LIN {X 0,Y 517.674,Z 1252.687,A -85,B 0,C 180,E1 12065.696,E2 12065.696} C_VEL
LIN {X 0,Y 518.294,Z 1242.725,A -85,B 0,C 180,E1 12070.089,E2 12070.089} C_VEL
LIN {X 0,Y 519.672,Z 1227.061,A -85,B 0,C 180,E1 12074.336,E2 12074.336} C_VEL
LIN {X 0,Y 522.079,Z 1206.878,A -85,B 0,C 180,E1 12078.165,E2 12078.165} C_VEL
LIN {X 0,Y 525.156,Z 1182.716,A -85,B 0,C 180,E1 12081.57,E2 12081.57} C_VEL
LIN {X 0,Y 529.072,Z 1152.709,A -85,B 0,C 180,E1 12084.747,E2 12084.747} C_VEL
LIN {X 0,Y 533.272,Z 1118.155,A -85,B 0,C 180,E1 12087.469,E2 12087.469} C_VEL
LIN {X 0,Y 537.249,Z 1080.299,A -85,B 0,C 180,E1 12089.617,E2 12089.617} C_VEL
LIN {X 0,Y 540.035,Z 1039.368,A -85,B 0,C 180,E1 12091.243,E2 12091.243} C_VEL
LIN {X 0,Y 532.268,Z 1011.624,A -85,B 0,C 180,E1 12092.744,E2 12092.744} C_VEL
LIN {X 0,Y 521.045,Z 988.142,A -85,B 0,C 180,E1 12094.497,E2 12094.497} C_VEL
LIN {X 0,Y 515.944,Z 978.381,A -85,B 0,C 180,E1 12095.418,E2 12095.418} C_VEL
LIN {X 0,Y 515.906,Z 977.53,A -85,B 0,C 180,E1 12095.954,E2 12095.954} C_VEL
LIN {X 0,Y 515.706,Z 977.53,A -85,B 0,C 180,E1 12102.493,E2 12102.493} C_VEL
LIN {X 0,Y 515.702,Z 977.53,A -85,B 0,C 180,E1 12107.495,E2 12107.495} C_VEL
LIN {X 0,Y 515.966,Z 977.849,A -85,B 0,C 180,E1 12113.885,E2 12113.885} C_VEL
LIN {X 0,Y 518.775,Z 983.54,A -85,B 0,C 180,E1 12114.433,E2 12114.433} C_VEL
LIN {X 0,Y 525.544,Z 1003.125,A -85,B 0,C 180,E1 12115.774,E2 12115.774} C_VEL
LIN {X 0,Y 540.092,Z 1052.552,A -85,B 0,C 180,E1 12118.245,E2 12118.245} C_VEL
LIN {X 0,Y 536.809,Z 1095.974,A -85,B 0,C 180,E1 12119.472,E2 12119.472} C_VEL
LIN {X 0,Y 533.589,Z 1130.82,A -85,B 0,C 180,E1 12120.973,E2 12120.973} C_VEL
LIN {X 0,Y 528.491,Z 1146.473,A -85,B 0,C 180,E1 12121.634,E2 12121.634} C_VEL
LIN {X 0,Y 523.112,Z 1161.648,A -85,B 0,C 180,E1 12122.384,E2 12122.384} C_VEL
LIN {X 0,Y 518.929,Z 1197.704,A -85,B 0,C 180,E1 12125.22,E2 12125.22} C_VEL
LIN {X 0,Y 515.24,Z 1230.103,A -85,B 0,C 180,E1 12128.666,E2 12128.666} C_VEL
LIN {X 0,Y 512.446,Z 1256.091,A -85,B 0,C 180,E1 12132.365,E2 12132.365} C_VEL
LIN {X 0,Y 510.731,Z 1276.42,A -85,B 0,C 180,E1 12136.278,E2 12136.278} C_VEL
LIN {X 0,Y 509.918,Z 1290.852,A -85,B 0,C 180,E1 12140.17,E2 12140.17} C_VEL
LIN {X 0,Y 509.696,Z 1300.49,A -85,B 0,C 180,E1 12144.192,E2 12144.192} C_VEL
LIN {X 0,Y 509.653,Z 1305.171,A -85,B 0,C 180,E1 12148.304,E2 12148.304} C_VEL
LIN {X 0,Y 509.652,Z 1305.175,A -85,B 0,C 180,E1 12151.712,E2 12151.712} C_VEL
LIN {X 0,Y 509.706,Z 1300.635,A -85,B 0,C 180,E1 12155.817,E2 12155.817} C_VEL
LIN {X 0,Y 509.891,Z 1291.146,A -85,B 0,C 180,E1 12159.847,E2 12159.847} C_VEL
LIN {X 0,Y 510.92,Z 1274.891,A -85,B 0,C 180,E1 12164.171,E2 12164.171} C_VEL
LIN {X 0,Y 512.738,Z 1253.925,A -85,B 0,C 180,E1 12168.086,E2 12168.086} C_VEL
LIN {X 0,Y 515.486,Z 1228.889,A -85,B 0,C 180,E1 12171.566,E2 12171.566} C_VEL
LIN {X 0,Y 518.975,Z 1198.242,A -85,B 0,C 180,E1 12174.779,E2 12174.779} C_VEL
LIN {X 0,Y 522.964,Z 1163.212,A -85,B 0,C 180,E1 12177.511,E2 12177.511} C_VEL
LIN {X 0,Y 526.968,Z 1123.902,A -85,B 0,C 180,E1 12179.713,E2 12179.713} C_VEL
LIN {X 0,Y 530.27,Z 1082.204,A -85,B 0,C 180,E1 12181.246,E2 12181.246} C_VEL
LIN {X 0,Y 531.189,Z 1051.195,A -85,B 0,C 180,E1 12181.983,E2 12181.983} C_VEL
LIN {X 0,Y 517.798,Z 1008.08,A -85,B 0,C 180,E1 12183.613,E2 12183.613} C_VEL
LIN {X 0,Y 514.673,Z 999.311,A -85,B 0,C 180,E1 12184.192,E2 12184.192} C_VEL
LIN {X 0,Y 508,Z 977.53,A -85,B 0,C 180,E1 12186.479,E2 12186.479} C_VEL
LIN {X 0,Y 507.893,Z 977.53,A -85,B 0,C 180,E1 12193.34,E2 12193.34} C_VEL
LIN {X 0,Y 507.84,Z 977.53,A -85,B 0,C 180,E1 12198.994,E2 12198.994} C_VEL
LIN {X 0,Y 507.949,Z 977.53,A -85,B 0,C 180,E1 12205.493,E2 12205.493} C_VEL
LIN {X 0,Y 508.183,Z 977.53,A -85,B 0,C 180,E1 12211.523,E2 12211.523} C_VEL
LIN {X 0,Y 508.423,Z 977.53,A -85,B 0,C 180,E1 12217.523,E2 12217.523} C_VEL
LIN {X 0,Y 508.509,Z 977.53,A -85,B 0,C 180,E1 12222.678,E2 12222.678} C_VEL
LIN {X 0,Y 508.671,Z 977.53,A -85,B 0,C 180,E1 12227.331,E2 12227.331} C_VEL
LIN {X 0,Y 523.418,Z 1014.68,A -85,B 0,C 180,E1 12229.87,E2 12229.87} C_VEL
LIN {X 0,Y 525.734,Z 1025.014,A -85,B 0,C 180,E1 12230.378,E2 12230.378} C_VEL
LIN {X 0,Y 522.592,Z 1078.23,A -85,B 0,C 180,E1 12231.992,E2 12231.992} C_VEL
LIN {X 0,Y 520.54,Z 1106.529,A -85,B 0,C 180,E1 12233.536,E2 12233.536} C_VEL
LIN {X 0,Y 517.847,Z 1132.303,A -85,B 0,C 180,E1 12235.712,E2 12235.712} C_VEL
LIN {X 0,Y 515.412,Z 1152.921,A -85,B 0,C 180,E1 12238.328,E2 12238.328} C_VEL
LIN {X 0,Y 513.42,Z 1168.559,A -85,B 0,C 180,E1 12241.28,E2 12241.28} C_VEL
LIN {X 0,Y 511.998,Z 1178.408,A -85,B 0,C 180,E1 12244.255,E2 12244.255} C_VEL
LIN {X 0,Y 511.229,Z 1182.945,A -85,B 0,C 180,E1 12246.82,E2 12246.82} C_VEL
LIN {X 0,Y 510.828,Z 1183.897,A -85,B 0,C 180,E1 12250.263,E2 12250.263} C_VEL
LIN {X 0,Y 511.052,Z 1178.841,A -85,B 0,C 180,E1 12253.732,E2 12253.732} C_VEL
LIN {X 0,Y 511.596,Z 1169.023,A -85,B 0,C 180,E1 12256.795,E2 12256.795} C_VEL
LIN {X 0,Y 512.738,Z 1152.99,A -85,B 0,C 180,E1 12259.878,E2 12259.878} C_VEL
LIN {X 0,Y 514.329,Z 1132.205,A -85,B 0,C 180,E1 12262.529,E2 12262.529} C_VEL
LIN {X 0,Y 515.926,Z 1107.861,A -85,B 0,C 180,E1 12264.663,E2 12264.663} C_VEL
LIN {X 0,Y 517.508,Z 1079.704,A -85,B 0,C 180,E1 12266.286,E2 12266.286} C_VEL
LIN {X 0,Y 518.405,Z 1049.368,A -85,B 0,C 180,E1 12267.293,E2 12267.293} C_VEL
LIN {X 0,Y 518.622,Z 1015.217,A -85,B 0,C 180,E1 12268.017,E2 12268.017} C_VEL
LIN {X 0,Y 508.273,Z 977.53,A -85,B 0,C 180,E1 12269.286,E2 12269.286} C_VEL
LIN {X 0,Y 507.992,Z 977.53,A -85,B 0,C 180,E1 12274.533,E2 12274.533} C_VEL
LIN {X 0,Y 507.906,Z 977.53,A -85,B 0,C 180,E1 12281.031,E2 12281.031} C_VEL
LIN {X 0,Y 507.88,Z 977.53,A -85,B 0,C 180,E1 12286.659,E2 12286.659} C_VEL
LIN {X 0,Y 507.922,Z 977.53,A -85,B 0,C 180,E1 12293.36,E2 12293.36} C_VEL
LIN {X 0,Y 508.127,Z 977.53,A -85,B 0,C 180,E1 12299.872,E2 12299.872} C_VEL
LIN {X 0,Y 508.284,Z 977.53,A -85,B 0,C 180,E1 12305.323,E2 12305.323} C_VEL
LIN {X 0,Y 508.485,Z 977.53,A -85,B 0,C 180,E1 12310.857,E2 12310.857} C_VEL
LIN {X 0,Y 508.621,Z 977.53,A -85,B 0,C 180,E1 12316.204,E2 12316.204} C_VEL
LIN {X 0,Y 508.884,Z 977.53,A -85,B 0,C 180,E1 12321.43,E2 12321.43} C_VEL
LIN {X 0,Y 509.137,Z 977.53,A -85,B 0,C 180,E1 12326.58,E2 12326.58} C_VEL
LIN {X 0,Y 509.259,Z 977.53,A -85,B 0,C 180,E1 12331.697,E2 12331.697} C_VEL
LIN {X 0,Y 508.941,Z 977.53,A -85,B 0,C 180,E1 12336.832,E2 12336.832} C_VEL
LIN {X 0,Y 508.71,Z 977.53,A -85,B 0,C 180,E1 12342.027,E2 12342.027} C_VEL
LIN {X 0,Y 508.514,Z 977.53,A -85,B 0,C 180,E1 12347.516,E2 12347.516} C_VEL
LIN {X 0,Y 508.315,Z 977.53,A -85,B 0,C 180,E1 12352.792,E2 12352.792} C_VEL
LIN {X 0,Y 508.162,Z 977.53,A -85,B 0,C 180,E1 12358.487,E2 12358.487} C_VEL
LIN {X 0,Y 508.026,Z 977.53,A -85,B 0,C 180,E1 12364.511,E2 12364.511} C_VEL
LIN {X 0,Y 507.876,Z 977.53,A -85,B 0,C 180,E1 12371.014,E2 12371.014} C_VEL
LIN {X 0,Y 507.861,Z 977.53,A -85,B 0,C 180,E1 12376.657,E2 12376.657} C_VEL
LIN {X 0,Y 507.925,Z 977.53,A -85,B 0,C 180,E1 12383.36,E2 12383.36} C_VEL
LIN {X 0,Y 508.032,Z 978.194,A -85,B 0,C 180,E1 12385.954,E2 12385.954} C_VEL
LIN {X 0,Y 527.737,Z 1030.087,A -85,B 0,C 180,E1 12388.197,E2 12388.197} C_VEL
LIN {X 0,Y 531.315,Z 1043.411,A -85,B 0,C 180,E1 12388.828,E2 12388.828} C_VEL
LIN {X 0,Y 528.029,Z 1082.986,A -85,B 0,C 180,E1 12390.438,E2 12390.438} C_VEL
LIN {X 0,Y 524.301,Z 1119.193,A -85,B 0,C 180,E1 12392.576,E2 12392.576} C_VEL
LIN {X 0,Y 520.228,Z 1153.562,A -85,B 0,C 180,E1 12395.352,E2 12395.352} C_VEL
LIN {X 0,Y 516.414,Z 1184.3,A -85,B 0,C 180,E1 12398.699,E2 12398.699} C_VEL
LIN {X 0,Y 513.431,Z 1209.4,A -85,B 0,C 180,E1 12402.381,E2 12402.381} C_VEL
LIN {X 0,Y 511.332,Z 1228.999,A -85,B 0,C 180,E1 12406.276,E2 12406.276} C_VEL
LIN {X 0,Y 510.227,Z 1242.925,A -85,B 0,C 180,E1 12410.157,E2 12410.157} C_VEL
LIN {X 0,Y 509.643,Z 1252.599,A -85,B 0,C 180,E1 12414.386,E2 12414.386} C_VEL
LIN {X 0,Y 509.472,Z 1256.861,A -85,B 0,C 180,E1 12418.284,E2 12418.284} C_VEL
LIN {X 0,Y 509.615,Z 1257.126,A -85,B 0,C 180,E1 12421.691,E2 12421.691} C_VEL
LIN {X 0,Y 509.798,Z 1253.133,A -85,B 0,C 180,E1 12425.784,E2 12425.784} C_VEL
LIN {X 0,Y 510.486,Z 1243.205,A -85,B 0,C 180,E1 12430.245,E2 12430.245} C_VEL
LIN {X 0,Y 511.978,Z 1227.568,A -85,B 0,C 180,E1 12434.556,E2 12434.556} C_VEL
LIN {X 0,Y 514.503,Z 1207.42,A -85,B 0,C 180,E1 12438.442,E2 12438.442} C_VEL
LIN {X 0,Y 517.774,Z 1183.304,A -85,B 0,C 180,E1 12441.893,E2 12441.893} C_VEL
LIN {X 0,Y 521.754,Z 1154.531,A -85,B 0,C 180,E1 12445.003,E2 12445.003} C_VEL
LIN {X 0,Y 526.022,Z 1121.129,A -85,B 0,C 180,E1 12447.716,E2 12447.716} C_VEL
LIN {X 0,Y 530.34,Z 1082.747,A -85,B 0,C 180,E1 12449.983,E2 12449.983} C_VEL
LIN {X 0,Y 533.531,Z 1041.642,A -85,B 0,C 180,E1 12451.665,E2 12451.665} C_VEL
LIN {X 0,Y 526.215,Z 1014.699,A -85,B 0,C 180,E1 12453.206,E2 12453.206} C_VEL
LIN {X 0,Y 515.247,Z 991.599,A -85,B 0,C 180,E1 12455.064,E2 12455.064} C_VEL
LIN {X 0,Y 508.007,Z 978.135,A -85,B 0,C 180,E1 12456.523,E2 12456.523} C_VEL
LIN {X 0,Y 507.751,Z 977.53,A -85,B 0,C 180,E1 12461.761,E2 12461.761} C_VEL
LIN {X 0,Y 507.746,Z 977.53,A -85,B 0,C 180,E1 12468.225,E2 12468.225} C_VEL
LIN {X 0,Y 508.045,Z 978.12,A -85,B 0,C 180,E1 12472.78,E2 12472.78} C_VEL
LIN {X 0,Y 510.907,Z 983.645,A -85,B 0,C 180,E1 12473.42,E2 12473.42} C_VEL
LIN {X 0,Y 516.711,Z 995.396,A -85,B 0,C 180,E1 12474.578,E2 12474.578} C_VEL
LIN {X 0,Y 529.642,Z 1040.211,A -85,B 0,C 180,E1 12477.114,E2 12477.114} C_VEL
LIN {X 0,Y 533.412,Z 1056.815,A -85,B 0,C 180,E1 12477.858,E2 12477.858} C_VEL
LIN {X 0,Y 529.842,Z 1098.874,A -85,B 0,C 180,E1 12479.135,E2 12479.135} C_VEL
LIN {X 0,Y 525.642,Z 1140.038,A -85,B 0,C 180,E1 12481.057,E2 12481.057} C_VEL
LIN {X 0,Y 523.112,Z 1161.648,A -85,B 0,C 180,E1 12482.384,E2 12482.384} C_VEL
LIN {X 0,Y 517.813,Z 1176.433,A -85,B 0,C 180,E1 12483.252,E2 12483.252} C_VEL
LIN {X 0,Y 512.524,Z 1190.574,A -85,B 0,C 180,E1 12484.236,E2 12484.236} C_VEL
LIN {X 0,Y 508.556,Z 1222.098,A -85,B 0,C 180,E1 12487.419,E2 12487.419} C_VEL
LIN {X 0,Y 505.44,Z 1248.801,A -85,B 0,C 180,E1 12490.981,E2 12490.981} C_VEL
LIN {X 0,Y 503.279,Z 1271.003,A -85,B 0,C 180,E1 12494.957,E2 12494.957} C_VEL
LIN {X 0,Y 502.25,Z 1287.239,A -85,B 0,C 180,E1 12498.997,E2 12498.997} C_VEL
LIN {X 0,Y 501.842,Z 1298.125,A -85,B 0,C 180,E1 12503.071,E2 12503.071} C_VEL
LIN {X 0,Y 501.743,Z 1303.439,A -85,B 0,C 180,E1 12506.545,E2 12506.545} C_VEL
LIN {X 0,Y 501.817,Z 1305.231,A -85,B 0,C 180,E1 12510.008,E2 12510.008} C_VEL
LIN {X 0,Y 501.751,Z 1303.45,A -85,B 0,C 180,E1 12513.471,E2 12513.471} C_VEL
LIN {X 0,Y 501.895,Z 1296.291,A -85,B 0,C 180,E1 12517.816,E2 12517.816} C_VEL
LIN {X 0,Y 502.37,Z 1284.818,A -85,B 0,C 180,E1 12521.752,E2 12521.752} C_VEL
LIN {X 0,Y 503.599,Z 1267.795,A -85,B 0,C 180,E1 12525.738,E2 12525.738} C_VEL
LIN {X 0,Y 505.82,Z 1245.102,A -85,B 0,C 180,E1 12529.593,E2 12529.593} C_VEL
LIN {X 0,Y 509.094,Z 1217.26,A -85,B 0,C 180,E1 12533.119,E2 12533.119} C_VEL
LIN {X 0,Y 513.025,Z 1185.22,A -85,B 0,C 180,E1 12536.165,E2 12536.165} C_VEL
LIN {X 0,Y 517.218,Z 1148.71,A -85,B 0,C 180,E1 12538.73,E2 12538.73} C_VEL
LIN {X 0,Y 521.122,Z 1108.432,A -85,B 0,C 180,E1 12540.705,E2 12540.705} C_VEL
LIN {X 0,Y 524.064,Z 1067.991,A -85,B 0,C 180,E1 12541.97,E2 12541.97} C_VEL
LIN {X 0,Y 524.17,Z 1053.575,A -85,B 0,C 180,E1 12542.301,E2 12542.301} C_VEL
LIN {X 0,Y 511.11,Z 1009.867,A -85,B 0,C 180,E1 12544.118,E2 12544.118} C_VEL
LIN {X 0,Y 506.989,Z 999.295,A -85,B 0,C 180,E1 12544.777,E2 12544.777} C_VEL
LIN {X 0,Y 499.999,Z 977.53,A -85,B 0,C 180,E1 12547.199,E2 12547.199} C_VEL
LIN {X 0,Y 499.992,Z 977.53,A -85,B 0,C 180,E1 12553.362,E2 12553.362} C_VEL
LIN {X 0,Y 499.925,Z 977.53,A -85,B 0,C 180,E1 12559.278,E2 12559.278} C_VEL
LIN {X 0,Y 499.99,Z 977.53,A -85,B 0,C 180,E1 12564.925,E2 12564.925} C_VEL
LIN {X 0,Y 500.282,Z 977.53,A -85,B 0,C 180,E1 12571.462,E2 12571.462} C_VEL
LIN {X 0,Y 500.418,Z 977.53,A -85,B 0,C 180,E1 12576.835,E2 12576.835} C_VEL
LIN {X 0,Y 500.589,Z 977.53,A -85,B 0,C 180,E1 12582.396,E2 12582.396} C_VEL
LIN {X 0,Y 500.704,Z 977.53,A -85,B 0,C 180,E1 12586.562,E2 12586.562} C_VEL
LIN {X 0,Y 515.66,Z 1013.787,A -85,B 0,C 180,E1 12589.264,E2 12589.264} C_VEL
LIN {X 0,Y 519.045,Z 1025.531,A -85,B 0,C 180,E1 12589.925,E2 12589.925} C_VEL
LIN {X 0,Y 515.519,Z 1080.567,A -85,B 0,C 180,E1 12591.668,E2 12591.668} C_VEL
LIN {X 0,Y 513.338,Z 1108.269,A -85,B 0,C 180,E1 12593.232,E2 12593.232} C_VEL
LIN {X 0,Y 510.608,Z 1132.606,A -85,B 0,C 180,E1 12595.332,E2 12595.332} C_VEL
LIN {X 0,Y 508.24,Z 1151.859,A -85,B 0,C 180,E1 12597.734,E2 12597.734} C_VEL
LIN {X 0,Y 506.21,Z 1166.874,A -85,B 0,C 180,E1 12600.441,E2 12600.441} C_VEL
LIN {X 0,Y 504.33,Z 1178.893,A -85,B 0,C 180,E1 12603.888,E2 12603.888} C_VEL
LIN {X 0,Y 503.389,Z 1184.19,A -85,B 0,C 180,E1 12606.927,E2 12606.927} C_VEL
LIN {X 0,Y 502.984,Z 1184.754,A -85,B 0,C 180,E1 12610.425,E2 12610.425} C_VEL
LIN {X 0,Y 503.256,Z 1179.276,A -85,B 0,C 180,E1 12613.949,E2 12613.949} C_VEL
LIN {X 0,Y 503.839,Z 1169.076,A -85,B 0,C 180,E1 12617.062,E2 12617.062} C_VEL
LIN {X 0,Y 504.987,Z 1152.489,A -85,B 0,C 180,E1 12620.197,E2 12620.197} C_VEL
LIN {X 0,Y 506.759,Z 1131.113,A -85,B 0,C 180,E1 12622.885,E2 12622.885} C_VEL
LIN {X 0,Y 508.43,Z 1106.223,A -85,B 0,C 180,E1 12625.023,E2 12625.023} C_VEL
LIN {X 0,Y 509.947,Z 1077.883,A -85,B 0,C 180,E1 12626.617,E2 12626.617} C_VEL
LIN {X 0,Y 510.834,Z 1047.342,A -85,B 0,C 180,E1 12627.591,E2 12627.591} C_VEL
LIN {X 0,Y 510.968,Z 1016.192,A -85,B 0,C 180,E1 12628.271,E2 12628.271} C_VEL
LIN {X 0,Y 500.334,Z 977.53,A -85,B 0,C 180,E1 12629.599,E2 12629.599} C_VEL
LIN {X 0,Y 500.034,Z 977.53,A -85,B 0,C 180,E1 12635.163,E2 12635.163} C_VEL
LIN {X 0,Y 500.026,Z 977.53,A -85,B 0,C 180,E1 12641.822,E2 12641.822} C_VEL
LIN {X 0,Y 499.982,Z 977.53,A -85,B 0,C 180,E1 12648.173,E2 12648.173} C_VEL
LIN {X 0,Y 500.008,Z 977.53,A -85,B 0,C 180,E1 12654.92,E2 12654.92} C_VEL
LIN {X 0,Y 500.265,Z 977.53,A -85,B 0,C 180,E1 12661.462,E2 12661.462} C_VEL
LIN {X 0,Y 500.393,Z 977.53,A -85,B 0,C 180,E1 12666.809,E2 12666.809} C_VEL
LIN {X 0,Y 500.609,Z 977.53,A -85,B 0,C 180,E1 12672.373,E2 12672.373} C_VEL
LIN {X 0,Y 500.777,Z 977.53,A -85,B 0,C 180,E1 12677.763,E2 12677.763} C_VEL
LIN {X 0,Y 501.074,Z 977.53,A -85,B 0,C 180,E1 12683.044,E2 12683.044} C_VEL
LIN {X 0,Y 501.241,Z 977.53,A -85,B 0,C 180,E1 12688.26,E2 12688.26} C_VEL
LIN {X 0,Y 501.19,Z 977.53,A -85,B 0,C 180,E1 12693.805,E2 12693.805} C_VEL
LIN {X 0,Y 500.897,Z 977.53,A -85,B 0,C 180,E1 12698.691,E2 12698.691} C_VEL
LIN {X 0,Y 500.67,Z 977.53,A -85,B 0,C 180,E1 12704.403,E2 12704.403} C_VEL
LIN {X 0,Y 500.51,Z 977.53,A -85,B 0,C 180,E1 12710.181,E2 12710.181} C_VEL
LIN {X 0,Y 500.295,Z 977.53,A -85,B 0,C 180,E1 12715.08,E2 12715.08} C_VEL
LIN {X 0,Y 500.138,Z 977.53,A -85,B 0,C 180,E1 12720.991,E2 12720.991} C_VEL
LIN {X 0,Y 499.975,Z 977.53,A -85,B 0,C 180,E1 12727.3,E2 12727.3} C_VEL
LIN {X 0,Y 499.98,Z 977.53,A -85,B 0,C 180,E1 12733.324,E2 12733.324} C_VEL
LIN {X 0,Y 499.918,Z 977.53,A -85,B 0,C 180,E1 12739.254,E2 12739.254} C_VEL
LIN {X 0,Y 500.1,Z 977.623,A -85,B 0,C 180,E1 12745.469,E2 12745.469} C_VEL
LIN {X 0,Y 519.896,Z 1030.125,A -85,B 0,C 180,E1 12747.782,E2 12747.782} C_VEL
LIN {X 0,Y 524.098,Z 1044.938,A -85,B 0,C 180,E1 12748.51,E2 12748.51} C_VEL
LIN {X 0,Y 520.714,Z 1083.85,A -85,B 0,C 180,E1 12750.125,E2 12750.125} C_VEL
LIN {X 0,Y 516.741,Z 1121.002,A -85,B 0,C 180,E1 12752.365,E2 12752.365} C_VEL
LIN {X 0,Y 512.524,Z 1155.393,A -85,B 0,C 180,E1 12755.215,E2 12755.215} C_VEL
LIN {X 0,Y 508.649,Z 1185.551,A -85,B 0,C 180,E1 12758.586,E2 12758.586} C_VEL
LIN {X 0,Y 505.597,Z 1210.485,A -85,B 0,C 180,E1 12762.325,E2 12762.325} C_VEL
LIN {X 0,Y 503.568,Z 1229.03,A -85,B 0,C 180,E1 12766.06,E2 12766.06} C_VEL
LIN {X 0,Y 502.397,Z 1243.094,A -85,B 0,C 180,E1 12770.002,E2 12770.002} C_VEL
LIN {X 0,Y 501.798,Z 1252.198,A -85,B 0,C 180,E1 12773.921,E2 12773.921} C_VEL
LIN {X 0,Y 501.579,Z 1257.214,A -85,B 0,C 180,E1 12778.257,E2 12778.257} C_VEL
LIN {X 0,Y 501.724,Z 1257.545,A -85,B 0,C 180,E1 12781.718,E2 12781.718} C_VEL
LIN {X 0,Y 501.932,Z 1253.311,A -85,B 0,C 180,E1 12786.052,E2 12786.052} C_VEL
LIN {X 0,Y 502.7,Z 1243.714,A -85,B 0,C 180,E1 12790.406,E2 12790.406} C_VEL
LIN {X 0,Y 504.275,Z 1228.116,A -85,B 0,C 180,E1 12794.783,E2 12794.783} C_VEL
LIN {X 0,Y 506.952,Z 1208.018,A -85,B 0,C 180,E1 12798.727,E2 12798.727} C_VEL
LIN {X 0,Y 510.417,Z 1183.973,A -85,B 0,C 180,E1 12802.225,E2 12802.225} C_VEL
LIN {X 0,Y 514.611,Z 1155.324,A -85,B 0,C 180,E1 12805.374,E2 12805.374} C_VEL
LIN {X 0,Y 519.16,Z 1121.878,A -85,B 0,C 180,E1 12808.136,E2 12808.136} C_VEL
LIN {X 0,Y 523.764,Z 1083.211,A -85,B 0,C 180,E1 12810.459,E2 12810.459} C_VEL
LIN {X 0,Y 526.921,Z 1042.452,A -85,B 0,C 180,E1 12812.187,E2 12812.187} C_VEL
LIN {X 0,Y 519.918,Z 1016.826,A -85,B 0,C 180,E1 12813.76,E2 12813.76} C_VEL
LIN {X 0,Y 509.535,Z 994.865,A -85,B 0,C 180,E1 12815.67,E2 12815.67} C_VEL
LIN {X 0,Y 502.475,Z 983.287,A -85,B 0,C 180,E1 12817.181,E2 12817.181} C_VEL
LIN {X 0,Y 499.956,Z 977.901,A -85,B 0,C 180,E1 12817.878,E2 12817.878} C_VEL
LIN {X 0,Y 499.824,Z 977.53,A -85,B 0,C 180,E1 12824.184,E2 12824.184} C_VEL
LIN {X 0,Y 499.892,Z 977.53,A -85,B 0,C 180,E1 12830.476,E2 12830.476} C_VEL
LIN {X 0,Y 500.005,Z 978.235,A -85,B 0,C 180,E1 12831.423,E2 12831.423} C_VEL
LIN {X 0,Y 503.017,Z 983.675,A -85,B 0,C 180,E1 12832.221,E2 12832.221} C_VEL
LIN {X 0,Y 511.284,Z 998.417,A -85,B 0,C 180,E1 12834.011,E2 12834.011} C_VEL
LIN {X 0,Y 523.258,Z 1041.663,A -85,B 0,C 180,E1 12836.591,E2 12836.591} C_VEL
LIN {X 0,Y 526.926,Z 1058.458,A -85,B 0,C 180,E1 12837.394,E2 12837.394} C_VEL
LIN {X 0,Y 523.013,Z 1100.851,A -85,B 0,C 180,E1 12838.742,E2 12838.742} C_VEL
LIN {X 0,Y 518.535,Z 1141.968,A -85,B 0,C 180,E1 12840.738,E2 12840.738} C_VEL
LIN {X 0,Y 513.979,Z 1179.263,A -85,B 0,C 180,E1 12843.292,E2 12843.292} C_VEL
LIN {X 0,Y 512.524,Z 1190.574,A -85,B 0,C 180,E1 12844.236,E2 12844.236} C_VEL
LIN {X 0,Y 507.109,Z 1204.205,A -85,B 0,C 180,E1 12845.327,E2 12845.327} C_VEL
LIN {X 0,Y 501.705,Z 1217.109,A -85,B 0,C 180,E1 12846.516,E2 12846.516} C_VEL
LIN {X 0,Y 498.124,Z 1245.562,A -85,B 0,C 180,E1 12850.228,E2 12850.228} C_VEL
LIN {X 0,Y 495.72,Z 1268.581,A -85,B 0,C 180,E1 12854.282,E2 12854.282} C_VEL
LIN {X 0,Y 494.413,Z 1286.258,A -85,B 0,C 180,E1 12858.635,E2 12858.635} C_VEL
LIN {X 0,Y 493.946,Z 1297.763,A -85,B 0,C 180,E1 12862.96,E2 12862.96} C_VEL
LIN {X 0,Y 493.856,Z 1303.072,A -85,B 0,C 180,E1 12866.49,E2 12866.49} C_VEL
LIN {X 0,Y 493.926,Z 1304.832,A -85,B 0,C 180,E1 12870.008,E2 12870.008} C_VEL
LIN {X 0,Y 493.829,Z 1302.415,A -85,B 0,C 180,E1 12874.129,E2 12874.129} C_VEL
LIN {X 0,Y 494.036,Z 1294.768,A -85,B 0,C 180,E1 12878.385,E2 12878.385} C_VEL
LIN {X 0,Y 494.733,Z 1280.939,A -85,B 0,C 180,E1 12882.838,E2 12882.838} C_VEL
LIN {X 0,Y 496.297,Z 1261.254,A -85,B 0,C 180,E1 12887.098,E2 12887.098} C_VEL
LIN {X 0,Y 498.997,Z 1237.037,A -85,B 0,C 180,E1 12890.913,E2 12890.913} C_VEL
LIN {X 0,Y 502.693,Z 1207.602,A -85,B 0,C 180,E1 12894.376,E2 12894.376} C_VEL
LIN {X 0,Y 506.726,Z 1174.921,A -85,B 0,C 180,E1 12897.26,E2 12897.26} C_VEL
LIN {X 0,Y 511.062,Z 1137.787,A -85,B 0,C 180,E1 12899.664,E2 12899.664} C_VEL
LIN {X 0,Y 514.859,Z 1096.916,A -85,B 0,C 180,E1 12901.489,E2 12901.489} C_VEL
LIN {X 0,Y 517.047,Z 1055.645,A -85,B 0,C 180,E1 12902.635,E2 12902.635} C_VEL
LIN {X 0,Y 504.776,Z 1012.446,A -85,B 0,C 180,E1 12904.605,E2 12904.605} C_VEL
LIN {X 0,Y 498.679,Z 997.453,A -85,B 0,C 180,E1 12905.61,E2 12905.61} C_VEL
LIN {X 0,Y 492.063,Z 977.53,A -85,B 0,C 180,E1 12908.026,E2 12908.026} C_VEL
LIN {X 0,Y 492.063,Z 977.53,A -85,B 0,C 180,E1 12912.657,E2 12912.657} C_VEL
LIN {X 0,Y 492.054,Z 977.53,A -85,B 0,C 180,E1 12917.665,E2 12917.665} C_VEL
LIN {X 0,Y 491.991,Z 977.53,A -85,B 0,C 180,E1 12924.205,E2 12924.205} C_VEL
LIN {X 0,Y 492.248,Z 977.53,A -85,B 0,C 180,E1 12930.512,E2 12930.512} C_VEL
LIN {X 0,Y 492.49,Z 977.53,A -85,B 0,C 180,E1 12936.44,E2 12936.44} C_VEL
LIN {X 0,Y 492.712,Z 977.53,A -85,B 0,C 180,E1 12942.459,E2 12942.459} C_VEL
LIN {X 0,Y 492.761,Z 977.613,A -85,B 0,C 180,E1 12945.725,E2 12945.725} C_VEL
LIN {X 0,Y 507.368,Z 1011.543,A -85,B 0,C 180,E1 12948.507,E2 12948.507} C_VEL
LIN {X 0,Y 512.187,Z 1028.95,A -85,B 0,C 180,E1 12949.542,E2 12949.542} C_VEL
LIN {X 0,Y 508.538,Z 1081.909,A -85,B 0,C 180,E1 12951.284,E2 12951.284} C_VEL
LIN {X 0,Y 506.127,Z 1110.036,A -85,B 0,C 180,E1 12952.919,E2 12952.919} C_VEL
LIN {X 0,Y 503.271,Z 1134.096,A -85,B 0,C 180,E1 12955.047,E2 12955.047} C_VEL
LIN {X 0,Y 500.495,Z 1154.757,A -85,B 0,C 180,E1 12957.743,E2 12957.743} C_VEL
LIN {X 0,Y 498.149,Z 1170.811,A -85,B 0,C 180,E1 12960.884,E2 12960.884} C_VEL
LIN {X 0,Y 496.368,Z 1181.461,A -85,B 0,C 180,E1 12964.389,E2 12964.389} C_VEL
LIN {X 0,Y 495.539,Z 1185.436,A -85,B 0,C 180,E1 12967.037,E2 12967.037} C_VEL
LIN {X 0,Y 495.154,Z 1185.542,A -85,B 0,C 180,E1 12970.592,E2 12970.592} C_VEL
LIN {X 0,Y 495.422,Z 1179.69,A -85,B 0,C 180,E1 12974.174,E2 12974.174} C_VEL
LIN {X 0,Y 496.17,Z 1168.057,A -85,B 0,C 180,E1 12977.563,E2 12977.563} C_VEL
LIN {X 0,Y 497.313,Z 1151.94,A -85,B 0,C 180,E1 12980.522,E2 12980.522} C_VEL
LIN {X 0,Y 499.209,Z 1129.928,A -85,B 0,C 180,E1 12983.251,E2 12983.251} C_VEL
LIN {X 0,Y 500.959,Z 1104.075,A -85,B 0,C 180,E1 12985.423,E2 12985.423} C_VEL
LIN {X 0,Y 502.468,Z 1075.953,A -85,B 0,C 180,E1 12986.958,E2 12986.958} C_VEL
LIN {X 0,Y 503.409,Z 1043.176,A -85,B 0,C 180,E1 12987.941,E2 12987.941} C_VEL
LIN {X 0,Y 503.447,Z 1017.654,A -85,B 0,C 180,E1 12988.515,E2 12988.515} C_VEL
LIN {X 0,Y 492.401,Z 977.53,A -85,B 0,C 180,E1 12989.936,E2 12989.936} C_VEL
LIN {X 0,Y 492.057,Z 977.53,A -85,B 0,C 180,E1 12996.794,E2 12996.794} C_VEL
LIN {X 0,Y 492.086,Z 977.53,A -85,B 0,C 180,E1 13002.655,E2 13002.655} C_VEL
LIN {X 0,Y 492.043,Z 977.53,A -85,B 0,C 180,E1 13007.665,E2 13007.665} C_VEL
LIN {X 0,Y 492.001,Z 977.53,A -85,B 0,C 180,E1 13014.176,E2 13014.176} C_VEL
LIN {X 0,Y 492.236,Z 977.53,A -85,B 0,C 180,E1 13020.484,E2 13020.484} C_VEL
LIN {X 0,Y 492.474,Z 977.53,A -85,B 0,C 180,E1 13026.414,E2 13026.414} C_VEL
LIN {X 0,Y 492.708,Z 977.53,A -85,B 0,C 180,E1 13032.454,E2 13032.454} C_VEL
LIN {X 0,Y 492.843,Z 977.53,A -85,B 0,C 180,E1 13037.563,E2 13037.563} C_VEL
LIN {X 0,Y 493.152,Z 977.53,A -85,B 0,C 180,E1 13042.932,E2 13042.932} C_VEL
LIN {X 0,Y 493.355,Z 977.53,A -85,B 0,C 180,E1 13048.232,E2 13048.232} C_VEL
LIN {X 0,Y 493.341,Z 977.53,A -85,B 0,C 180,E1 13053.514,E2 13053.514} C_VEL
LIN {X 0,Y 492.978,Z 977.53,A -85,B 0,C 180,E1 13058.832,E2 13058.832} C_VEL
LIN {X 0,Y 492.778,Z 977.53,A -85,B 0,C 180,E1 13064.232,E2 13064.232} C_VEL
LIN {X 0,Y 492.616,Z 977.53,A -85,B 0,C 180,E1 13069.768,E2 13069.768} C_VEL
LIN {X 0,Y 492.331,Z 977.53,A -85,B 0,C 180,E1 13075.514,E2 13075.514} C_VEL
LIN {X 0,Y 492.196,Z 977.53,A -85,B 0,C 180,E1 13081.548,E2 13081.548} C_VEL
LIN {X 0,Y 492.072,Z 977.53,A -85,B 0,C 180,E1 13088.005,E2 13088.005} C_VEL
LIN {X 0,Y 492.072,Z 977.53,A -85,B 0,C 180,E1 13092.634,E2 13092.634} C_VEL
LIN {X 0,Y 492.03,Z 977.53,A -85,B 0,C 180,E1 13097.643,E2 13097.643} C_VEL
LIN {X 0,Y 492.022,Z 977.53,A -85,B 0,C 180,E1 13104.177,E2 13104.177} C_VEL
LIN {X 0,Y 492.139,Z 977.53,A -85,B 0,C 180,E1 13104.989,E2 13104.989} C_VEL
LIN {X 0,Y 512.159,Z 1030.55,A -85,B 0,C 180,E1 13107.375,E2 13107.375} C_VEL
LIN {X 0,Y 516.773,Z 1047.714,A -85,B 0,C 180,E1 13108.232,E2 13108.232} C_VEL
LIN {X 0,Y 513.204,Z 1086.842,A -85,B 0,C 180,E1 13109.922,E2 13109.922} C_VEL
LIN {X 0,Y 509.048,Z 1124.404,A -85,B 0,C 180,E1 13112.273,E2 13112.273} C_VEL
LIN {X 0,Y 504.615,Z 1158.836,A -85,B 0,C 180,E1 13115.249,E2 13115.249} C_VEL
LIN {X 0,Y 500.682,Z 1188.432,A -85,B 0,C 180,E1 13118.694,E2 13118.694} C_VEL
LIN {X 0,Y 497.637,Z 1212.776,A -85,B 0,C 180,E1 13122.49,E2 13122.49} C_VEL
LIN {X 0,Y 495.437,Z 1232.615,A -85,B 0,C 180,E1 13126.728,E2 13126.728} C_VEL
LIN {X 0,Y 494.318,Z 1246.817,A -85,B 0,C 180,E1 13131.172,E2 13131.172} C_VEL
LIN {X 0,Y 493.791,Z 1255.09,A -85,B 0,C 180,E1 13135.537,E2 13135.537} C_VEL
LIN {X 0,Y 493.769,Z 1258.191,A -85,B 0,C 180,E1 13139.987,E2 13139.987} C_VEL
LIN {X 0,Y 493.858,Z 1256.883,A -85,B 0,C 180,E1 13143.505,E2 13143.505} C_VEL
LIN {X 0,Y 494.307,Z 1250.605,A -85,B 0,C 180,E1 13147.915,E2 13147.915} C_VEL
LIN {X 0,Y 495.488,Z 1238.763,A -85,B 0,C 180,E1 13152.347,E2 13152.347} C_VEL
LIN {X 0,Y 497.652,Z 1221.505,A -85,B 0,C 180,E1 13156.602,E2 13156.602} C_VEL
LIN {X 0,Y 500.774,Z 1199.915,A -85,B 0,C 180,E1 13160.433,E2 13160.433} C_VEL
LIN {X 0,Y 504.968,Z 1172.558,A -85,B 0,C 180,E1 13164.043,E2 13164.043} C_VEL
LIN {X 0,Y 509.998,Z 1139.291,A -85,B 0,C 180,E1 13167.292,E2 13167.292} C_VEL
LIN {X 0,Y 514.926,Z 1102.902,A -85,B 0,C 180,E1 13169.887,E2 13169.887} C_VEL
LIN {X 0,Y 519.41,Z 1064.543,A -85,B 0,C 180,E1 13171.839,E2 13171.839} C_VEL
LIN {X 0,Y 520.561,Z 1044.416,A -85,B 0,C 180,E1 13172.677,E2 13172.677} C_VEL
LIN {X 0,Y 513.932,Z 1019.448,A -85,B 0,C 180,E1 13174.306,E2 13174.306} C_VEL
LIN {X 0,Y 504.129,Z 998.823,A -85,B 0,C 180,E1 13176.273,E2 13176.273} C_VEL
LIN {X 0,Y 497.569,Z 988.1,A -85,B 0,C 180,E1 13177.813,E2 13177.813} C_VEL
LIN {X 0,Y 494.951,Z 983.678,A -85,B 0,C 180,E1 13178.57,E2 13178.57} C_VEL
LIN {X 0,Y 492.029,Z 978.397,A -85,B 0,C 180,E1 13179.589,E2 13179.589} C_VEL
LIN {X 0,Y 491.97,Z 977.53,A -85,B 0,C 180,E1 13180.278,E2 13180.278} C_VEL
LIN {X 0,Y 491.896,Z 977.53,A -85,B 0,C 180,E1 13185.089,E2 13185.089} C_VEL
LIN {X 0,Y 491.979,Z 978.308,A -85,B 0,C 180,E1 13189.643,E2 13189.643} C_VEL
LIN {X 0,Y 495.15,Z 983.796,A -85,B 0,C 180,E1 13190.748,E2 13190.748} C_VEL
LIN {X 0,Y 503.507,Z 997.303,A -85,B 0,C 180,E1 13192.889,E2 13192.889} C_VEL
LIN {X 0,Y 507.189,Z 1005.771,A -85,B 0,C 180,E1 13193.739,E2 13193.739} C_VEL
LIN {X 0,Y 518.647,Z 1050.506,A -85,B 0,C 180,E1 13196.419,E2 13196.419} C_VEL
LIN {X 0,Y 520.422,Z 1061.325,A -85,B 0,C 180,E1 13196.934,E2 13196.934} C_VEL
LIN {X 0,Y 516.021,Z 1105.004,A -85,B 0,C 180,E1 13198.417,E2 13198.417} C_VEL
LIN {X 0,Y 511.03,Z 1146.344,A -85,B 0,C 180,E1 13200.557,E2 13200.557} C_VEL
LIN {X 0,Y 506.23,Z 1183.12,A -85,B 0,C 180,E1 13203.21,E2 13203.21} C_VEL
LIN {X 0,Y 501.824,Z 1216.297,A -85,B 0,C 180,E1 13206.425,E2 13206.425} C_VEL
LIN {X 0,Y 501.705,Z 1217.109,A -85,B 0,C 180,E1 13206.516,E2 13206.516} C_VEL
LIN {X 0,Y 496.255,Z 1229.344,A -85,B 0,C 180,E1 13207.825,E2 13207.825} C_VEL
LIN {X 0,Y 491.029,Z 1240.799,A -85,B 0,C 180,E1 13209.242,E2 13209.242} C_VEL
LIN {X 0,Y 488.186,Z 1264.851,A -85,B 0,C 180,E1 13213.324,E2 13213.324} C_VEL
LIN {X 0,Y 486.712,Z 1282.415,A -85,B 0,C 180,E1 13217.421,E2 13217.421} C_VEL
LIN {X 0,Y 486.153,Z 1295.547,A -85,B 0,C 180,E1 13221.946,E2 13221.946} C_VEL
LIN {X 0,Y 485.955,Z 1302.713,A -85,B 0,C 180,E1 13226.433,E2 13226.433} C_VEL
LIN {X 0,Y 486.036,Z 1304.431,A -85,B 0,C 180,E1 13230.008,E2 13230.008} C_VEL
LIN {X 0,Y 485.942,Z 1302.104,A -85,B 0,C 180,E1 13234.067,E2 13234.067} C_VEL
LIN {X 0,Y 486.143,Z 1294.235,A -85,B 0,C 180,E1 13238.522,E2 13238.522} C_VEL
LIN {X 0,Y 486.889,Z 1280.259,A -85,B 0,C 180,E1 13243.048,E2 13243.048} C_VEL
LIN {X 0,Y 488.578,Z 1260.371,A -85,B 0,C 180,E1 13247.377,E2 13247.377} C_VEL
LIN {X 0,Y 491.41,Z 1235.909,A -85,B 0,C 180,E1 13251.251,E2 13251.251} C_VEL
LIN {X 0,Y 495.106,Z 1207.281,A -85,B 0,C 180,E1 13254.654,E2 13254.654} C_VEL
LIN {X 0,Y 499.385,Z 1173.578,A -85,B 0,C 180,E1 13257.658,E2 13257.658} C_VEL
LIN {X 0,Y 503.955,Z 1135.486,A -85,B 0,C 180,E1 13260.125,E2 13260.125} C_VEL
LIN {X 0,Y 507.823,Z 1094.549,A -85,B 0,C 180,E1 13261.93,E2 13261.93} C_VEL
LIN {X 0,Y 509.919,Z 1057.283,A -85,B 0,C 180,E1 13263.026,E2 13263.026} C_VEL
LIN {X 0,Y 499.263,Z 1016.91,A -85,B 0,C 180,E1 13265.002,E2 13265.002} C_VEL
LIN {X 0,Y 490.224,Z 995.351,A -85,B 0,C 180,E1 13266.55,E2 13266.55} C_VEL
LIN {X 0,Y 484.116,Z 977.53,A -85,B 0,C 180,E1 13268.867,E2 13268.867} C_VEL
LIN {X 0,Y 484.059,Z 977.53,A -85,B 0,C 180,E1 13273.973,E2 13273.973} C_VEL
LIN {X 0,Y 484.053,Z 977.53,A -85,B 0,C 180,E1 13278.923,E2 13278.923} C_VEL
LIN {X 0,Y 484.065,Z 977.53,A -85,B 0,C 180,E1 13284.491,E2 13284.491} C_VEL
LIN {X 0,Y 484.307,Z 977.53,A -85,B 0,C 180,E1 13289.979,E2 13289.979} C_VEL
LIN {X 0,Y 484.517,Z 977.53,A -85,B 0,C 180,E1 13296.028,E2 13296.028} C_VEL
LIN {X 0,Y 484.716,Z 977.53,A -85,B 0,C 180,E1 13301.799,E2 13301.799} C_VEL
LIN {X 0,Y 484.817,Z 977.829,A -85,B 0,C 180,E1 13304.817,E2 13304.817} C_VEL
LIN {X 0,Y 499.507,Z 1010.674,A -85,B 0,C 180,E1 13307.782,E2 13307.782} C_VEL
LIN {X 0,Y 505.541,Z 1030.595,A -85,B 0,C 180,E1 13309.082,E2 13309.082} C_VEL
LIN {X 0,Y 501.595,Z 1083.395,A -85,B 0,C 180,E1 13310.888,E2 13310.888} C_VEL
LIN {X 0,Y 499.147,Z 1110.474,A -85,B 0,C 180,E1 13312.491,E2 13312.491} C_VEL
LIN {X 0,Y 495.967,Z 1135.592,A -85,B 0,C 180,E1 13314.754,E2 13314.754} C_VEL
LIN {X 0,Y 493.108,Z 1155.623,A -85,B 0,C 180,E1 13317.417,E2 13317.417} C_VEL
LIN {X 0,Y 490.674,Z 1171.045,A -85,B 0,C 180,E1 13320.455,E2 13320.455} C_VEL
LIN {X 0,Y 488.943,Z 1181.047,A -85,B 0,C 180,E1 13323.566,E2 13323.566} C_VEL
LIN {X 0,Y 487.696,Z 1186.626,A -85,B 0,C 180,E1 13327.151,E2 13327.151} C_VEL
LIN {X 0,Y 487.318,Z 1186.329,A -85,B 0,C 180,E1 13330.764,E2 13330.764} C_VEL
LIN {X 0,Y 487.629,Z 1180.049,A -85,B 0,C 180,E1 13334.406,E2 13334.406} C_VEL
LIN {X 0,Y 488.433,Z 1167.95,A -85,B 0,C 180,E1 13337.851,E2 13337.851} C_VEL
LIN {X 0,Y 489.684,Z 1151.339,A -85,B 0,C 180,E1 13340.857,E2 13340.857} C_VEL
LIN {X 0,Y 491.52,Z 1129.603,A -85,B 0,C 180,E1 13343.524,E2 13343.524} C_VEL
LIN {X 0,Y 493.407,Z 1103.421,A -85,B 0,C 180,E1 13345.718,E2 13345.718} C_VEL
LIN {X 0,Y 494.937,Z 1074.285,A -85,B 0,C 180,E1 13347.283,E2 13347.283} C_VEL
LIN {X 0,Y 495.986,Z 1039.705,A -85,B 0,C 180,E1 13348.285,E2 13348.285} C_VEL
LIN {X 0,Y 496.041,Z 1019.546,A -85,B 0,C 180,E1 13348.753,E2 13348.753} C_VEL
LIN {X 0,Y 484.436,Z 977.53,A -85,B 0,C 180,E1 13350.283,E2 13350.283} C_VEL
LIN {X 0,Y 484.141,Z 977.53,A -85,B 0,C 180,E1 13356.499,E2 13356.499} C_VEL
LIN {X 0,Y 484.107,Z 977.53,A -85,B 0,C 180,E1 13361.293,E2 13361.293} C_VEL
LIN {X 0,Y 484.055,Z 977.53,A -85,B 0,C 180,E1 13366.463,E2 13366.463} C_VEL
LIN {X 0,Y 484.115,Z 977.53,A -85,B 0,C 180,E1 13371.501,E2 13371.501} C_VEL
LIN {X 0,Y 484.184,Z 977.53,A -85,B 0,C 180,E1 13377.848,E2 13377.848} C_VEL
LIN {X 0,Y 484.426,Z 977.53,A -85,B 0,C 180,E1 13384.02,E2 13384.02} C_VEL
LIN {X 0,Y 484.661,Z 977.53,A -85,B 0,C 180,E1 13389.876,E2 13389.876} C_VEL
LIN {X 0,Y 484.864,Z 977.53,A -85,B 0,C 180,E1 13395.673,E2 13395.673} C_VEL
LIN {X 0,Y 485.12,Z 977.53,A -85,B 0,C 180,E1 13401.007,E2 13401.007} C_VEL
LIN {X 0,Y 485.449,Z 977.53,A -85,B 0,C 180,E1 13406.413,E2 13406.413} C_VEL
LIN {X 0,Y 485.553,Z 977.53,A -85,B 0,C 180,E1 13411.78,E2 13411.78} C_VEL
LIN {X 0,Y 485.187,Z 977.53,A -85,B 0,C 180,E1 13417.168,E2 13417.168} C_VEL
LIN {X 0,Y 484.911,Z 977.53,A -85,B 0,C 180,E1 13422.626,E2 13422.626} C_VEL
LIN {X 0,Y 484.731,Z 977.53,A -85,B 0,C 180,E1 13428.207,E2 13428.207} C_VEL
LIN {X 0,Y 484.463,Z 977.53,A -85,B 0,C 180,E1 13433.982,E2 13433.982} C_VEL
LIN {X 0,Y 484.313,Z 977.53,A -85,B 0,C 180,E1 13440.029,E2 13440.029} C_VEL
LIN {X 0,Y 484.132,Z 977.53,A -85,B 0,C 180,E1 13446.479,E2 13446.479} C_VEL
LIN {X 0,Y 484.087,Z 977.53,A -85,B 0,C 180,E1 13451.291,E2 13451.291} C_VEL
LIN {X 0,Y 484.043,Z 977.53,A -85,B 0,C 180,E1 13456.462,E2 13456.462} C_VEL
LIN {X 0,Y 484.088,Z 977.53,A -85,B 0,C 180,E1 13463.496,E2 13463.496} C_VEL
LIN {X 0,Y 484.19,Z 977.825,A -85,B 0,C 180,E1 13464.505,E2 13464.505} C_VEL
LIN {X 0,Y 504.454,Z 1031.081,A -85,B 0,C 180,E1 13466.968,E2 13466.968} C_VEL
LIN {X 0,Y 509.521,Z 1049.091,A -85,B 0,C 180,E1 13467.899,E2 13467.899} C_VEL
LIN {X 0,Y 505.799,Z 1089.073,A -85,B 0,C 180,E1 13469.676,E2 13469.676} C_VEL
LIN {X 0,Y 501.294,Z 1127.569,A -85,B 0,C 180,E1 13472.174,E2 13472.174} C_VEL
LIN {X 0,Y 496.782,Z 1161.298,A -85,B 0,C 180,E1 13475.193,E2 13475.193} C_VEL
LIN {X 0,Y 492.914,Z 1189.612,A -85,B 0,C 180,E1 13478.579,E2 13478.579} C_VEL
LIN {X 0,Y 489.825,Z 1213.804,A -85,B 0,C 180,E1 13482.434,E2 13482.434} C_VEL
LIN {X 0,Y 487.659,Z 1232.608,A -85,B 0,C 180,E1 13486.512,E2 13486.512} C_VEL
LIN {X 0,Y 486.452,Z 1246.974,A -85,B 0,C 180,E1 13491.028,E2 13491.028} C_VEL
LIN {X 0,Y 485.899,Z 1255.574,A -85,B 0,C 180,E1 13495.606,E2 13495.606} C_VEL
LIN {X 0,Y 485.878,Z 1258.572,A -85,B 0,C 180,E1 13499.987,E2 13499.987} C_VEL
LIN {X 0,Y 485.976,Z 1256.974,A -85,B 0,C 180,E1 13503.964,E2 13503.964} C_VEL
LIN {X 0,Y 486.484,Z 1251.128,A -85,B 0,C 180,E1 13508.043,E2 13508.043} C_VEL
LIN {X 0,Y 487.732,Z 1239.349,A -85,B 0,C 180,E1 13512.546,E2 13512.546} C_VEL
LIN {X 0,Y 490.045,Z 1222.073,A -85,B 0,C 180,E1 13516.888,E2 13516.888} C_VEL
LIN {X 0,Y 493.433,Z 1200.309,A -85,B 0,C 180,E1 13520.81,E2 13520.81} C_VEL
LIN {X 0,Y 497.746,Z 1173.596,A -85,B 0,C 180,E1 13524.398,E2 13524.398} C_VEL
LIN {X 0,Y 502.988,Z 1141.099,A -85,B 0,C 180,E1 13527.65,E2 13527.65} C_VEL
LIN {X 0,Y 508.293,Z 1104.221,A -85,B 0,C 180,E1 13530.344,E2 13530.344} C_VEL
LIN {X 0,Y 513.155,Z 1065.355,A -85,B 0,C 180,E1 13532.366,E2 13532.366} C_VEL
LIN {X 0,Y 514.264,Z 1046.17,A -85,B 0,C 180,E1 13533.206,E2 13533.206} C_VEL
LIN {X 0,Y 508.138,Z 1022.333,A -85,B 0,C 180,E1 13534.87,E2 13534.87} C_VEL
LIN {X 0,Y 498.591,Z 1001.77,A -85,B 0,C 180,E1 13537.001,E2 13537.001} C_VEL
LIN {X 0,Y 491.402,Z 990.204,A -85,B 0,C 180,E1 13538.969,E2 13538.969} C_VEL
LIN {X 0,Y 487.815,Z 984.239,A -85,B 0,C 180,E1 13540.344,E2 13540.344} C_VEL
LIN {X 0,Y 484.109,Z 978.638,A -85,B 0,C 180,E1 13542.58,E2 13542.58} C_VEL
LIN {X 0,Y 483.926,Z 977.53,A -85,B 0,C 180,E1 13543.516,E2 13543.516} C_VEL
LIN {X 0,Y 483.977,Z 978.261,A -85,B 0,C 180,E1 13546.477,E2 13546.477} C_VEL
LIN {X 0,Y 487.927,Z 984.313,A -85,B 0,C 180,E1 13548.939,E2 13548.939} C_VEL
LIN {X 0,Y 493.762,Z 993.833,A -85,B 0,C 180,E1 13551.025,E2 13551.025} C_VEL
LIN {X 0,Y 501.573,Z 1007.116,A -85,B 0,C 180,E1 13552.999,E2 13552.999} C_VEL
LIN {X 0,Y 512.009,Z 1050.026,A -85,B 0,C 180,E1 13555.757,E2 13555.757} C_VEL
LIN {X 0,Y 514.217,Z 1062.345,A -85,B 0,C 180,E1 13556.405,E2 13556.405} C_VEL
LIN {X 0,Y 509.376,Z 1106.176,A -85,B 0,C 180,E1 13557.957,E2 13557.957} C_VEL
LIN {X 0,Y 504.068,Z 1147.297,A -85,B 0,C 180,E1 13560.15,E2 13560.15} C_VEL
LIN {X 0,Y 498.912,Z 1184.444,A -85,B 0,C 180,E1 13562.908,E2 13562.908} C_VEL
LIN {X 0,Y 494.14,Z 1218.096,A -85,B 0,C 180,E1 13566.281,E2 13566.281} C_VEL
LIN {X 0,Y 491.029,Z 1240.799,A -85,B 0,C 180,E1 13569.242,E2 13569.242} C_VEL
LIN {X 0,Y 485.994,Z 1251.489,A -85,B 0,C 180,E1 13570.764,E2 13570.764} C_VEL
LIN {X 0,Y 480.901,Z 1261.225,A -85,B 0,C 180,E1 13572.392,E2 13572.392} C_VEL
LIN {X 0,Y 479.028,Z 1280.419,A -85,B 0,C 180,E1 13576.751,E2 13576.751} C_VEL
LIN {X 0,Y 478.275,Z 1293.073,A -85,B 0,C 180,E1 13580.894,E2 13580.894} C_VEL
LIN {X 0,Y 478.121,Z 1300.151,A -85,B 0,C 180,E1 13584.553,E2 13584.553} C_VEL
LIN {X 0,Y 478.08,Z 1303.665,A -85,B 0,C 180,E1 13588.192,E2 13588.192} C_VEL
LIN {X 0,Y 478.108,Z 1303.51,A -85,B 0,C 180,E1 13591.825,E2 13591.825} C_VEL
LIN {X 0,Y 478.176,Z 1298.364,A -85,B 0,C 180,E1 13596.376,E2 13596.376} C_VEL
LIN {X 0,Y 478.454,Z 1288.769,A -85,B 0,C 180,E1 13600.501,E2 13600.501} C_VEL
LIN {X 0,Y 479.621,Z 1272.638,A -85,B 0,C 180,E1 13604.947,E2 13604.947} C_VEL
LIN {X 0,Y 481.686,Z 1252.265,A -85,B 0,C 180,E1 13608.937,E2 13608.937} C_VEL
LIN {X 0,Y 485.083,Z 1225.504,A -85,B 0,C 180,E1 13612.812,E2 13612.812} C_VEL
LIN {X 0,Y 489.142,Z 1194.524,A -85,B 0,C 180,E1 13616.167,E2 13616.167} C_VEL
LIN {X 0,Y 493.743,Z 1158.719,A -85,B 0,C 180,E1 13619.041,E2 13619.041} C_VEL
LIN {X 0,Y 498.206,Z 1119.762,A -85,B 0,C 180,E1 13621.258,E2 13621.258} C_VEL
LIN {X 0,Y 502.11,Z 1076.121,A -85,B 0,C 180,E1 13622.911,E2 13622.911} C_VEL
LIN {X 0,Y 503.199,Z 1059.089,A -85,B 0,C 180,E1 13623.485,E2 13623.485} C_VEL
LIN {X 0,Y 493.426,Z 1020.45,A -85,B 0,C 180,E1 13625.465,E2 13625.465} C_VEL
LIN {X 0,Y 482.445,Z 995.26,A -85,B 0,C 180,E1 13627.326,E2 13627.326} C_VEL
LIN {X 0,Y 476.243,Z 977.53,A -85,B 0,C 180,E1 13629.884,E2 13629.884} C_VEL
LIN {X 0,Y 476.104,Z 977.53,A -85,B 0,C 180,E1 13635.583,E2 13635.583} C_VEL
LIN {X 0,Y 476.096,Z 977.53,A -85,B 0,C 180,E1 13640.488,E2 13640.488} C_VEL
LIN {X 0,Y 476.217,Z 977.53,A -85,B 0,C 180,E1 13647.274,E2 13647.274} C_VEL
LIN {X 0,Y 476.475,Z 977.53,A -85,B 0,C 180,E1 13653.58,E2 13653.58} C_VEL
LIN {X 0,Y 476.742,Z 977.53,A -85,B 0,C 180,E1 13659.552,E2 13659.552} C_VEL
LIN {X 0,Y 476.89,Z 977.896,A -85,B 0,C 180,E1 13663.814,E2 13663.814} C_VEL
LIN {X 0,Y 491.795,Z 1009.98,A -85,B 0,C 180,E1 13667.022,E2 13667.022} C_VEL
LIN {X 0,Y 498.981,Z 1031.745,A -85,B 0,C 180,E1 13668.592,E2 13668.592} C_VEL
LIN {X 0,Y 494.781,Z 1083.888,A -85,B 0,C 180,E1 13670.428,E2 13670.428} C_VEL
LIN {X 0,Y 492.012,Z 1112.447,A -85,B 0,C 180,E1 13672.159,E2 13672.159} C_VEL
LIN {X 0,Y 488.683,Z 1137.145,A -85,B 0,C 180,E1 13674.453,E2 13674.453} C_VEL
LIN {X 0,Y 485.473,Z 1158.128,A -85,B 0,C 180,E1 13677.351,E2 13677.351} C_VEL
LIN {X 0,Y 482.922,Z 1173.155,A -85,B 0,C 180,E1 13680.462,E2 13680.462} C_VEL
LIN {X 0,Y 481.136,Z 1182.69,A -85,B 0,C 180,E1 13683.624,E2 13683.624} C_VEL
LIN {X 0,Y 479.839,Z 1187.792,A -85,B 0,C 180,E1 13687.269,E2 13687.269} C_VEL
LIN {X 0,Y 479.496,Z 1187.111,A -85,B 0,C 180,E1 13690.942,E2 13690.942} C_VEL
LIN {X 0,Y 479.83,Z 1180.362,A -85,B 0,C 180,E1 13694.645,E2 13694.645} C_VEL
LIN {X 0,Y 480.698,Z 1167.837,A -85,B 0,C 180,E1 13698.148,E2 13698.148} C_VEL
LIN {X 0,Y 482.055,Z 1150.616,A -85,B 0,C 180,E1 13701.203,E2 13701.203} C_VEL
LIN {X 0,Y 483.9,Z 1128.267,A -85,B 0,C 180,E1 13703.91,E2 13703.91} C_VEL
LIN {X 0,Y 485.812,Z 1102.655,A -85,B 0,C 180,E1 13706.022,E2 13706.022} C_VEL
LIN {X 0,Y 487.418,Z 1073.516,A -85,B 0,C 180,E1 13707.574,E2 13707.574} C_VEL
LIN {X 0,Y 488.567,Z 1035.251,A -85,B 0,C 180,E1 13708.657,E2 13708.657} C_VEL
LIN {X 0,Y 488.427,Z 1020.558,A -85,B 0,C 180,E1 13709.016,E2 13709.016} C_VEL
LIN {X 0,Y 476.499,Z 977.53,A -85,B 0,C 180,E1 13710.595,E2 13710.595} C_VEL
LIN {X 0,Y 476.184,Z 977.53,A -85,B 0,C 180,E1 13717.281,E2 13717.281} C_VEL
LIN {X 0,Y 476.128,Z 977.53,A -85,B 0,C 180,E1 13722.936,E2 13722.936} C_VEL
LIN {X 0,Y 476.078,Z 977.53,A -85,B 0,C 180,E1 13728.046,E2 13728.046} C_VEL
LIN {X 0,Y 476.185,Z 977.53,A -85,B 0,C 180,E1 13735.046,E2 13735.046} C_VEL
LIN {X 0,Y 476.426,Z 977.53,A -85,B 0,C 180,E1 13741.496,E2 13741.496} C_VEL
LIN {X 0,Y 476.657,Z 977.53,A -85,B 0,C 180,E1 13747.566,E2 13747.566} C_VEL
LIN {X 0,Y 476.864,Z 977.53,A -85,B 0,C 180,E1 13753.374,E2 13753.374} C_VEL
LIN {X 0,Y 477.121,Z 977.53,A -85,B 0,C 180,E1 13759.939,E2 13759.939} C_VEL
LIN {X 0,Y 477.538,Z 977.53,A -85,B 0,C 180,E1 13766.353,E2 13766.353} C_VEL
LIN {X 0,Y 477.663,Z 977.53,A -85,B 0,C 180,E1 13771.809,E2 13771.809} C_VEL
LIN {X 0,Y 477.263,Z 977.53,A -85,B 0,C 180,E1 13777.288,E2 13777.288} C_VEL
LIN {X 0,Y 477.006,Z 977.53,A -85,B 0,C 180,E1 13782.839,E2 13782.839} C_VEL
LIN {X 0,Y 476.787,Z 977.53,A -85,B 0,C 180,E1 13788.521,E2 13788.521} C_VEL
LIN {X 0,Y 476.532,Z 977.53,A -85,B 0,C 180,E1 13794.407,E2 13794.407} C_VEL
LIN {X 0,Y 476.306,Z 977.53,A -85,B 0,C 180,E1 13800.788,E2 13800.788} C_VEL
LIN {X 0,Y 476.17,Z 977.53,A -85,B 0,C 180,E1 13807.28,E2 13807.28} C_VEL
LIN {X 0,Y 476.112,Z 977.53,A -85,B 0,C 180,E1 13812.934,E2 13812.934} C_VEL
LIN {X 0,Y 476.061,Z 977.53,A -85,B 0,C 180,E1 13818.044,E2 13818.044} C_VEL
LIN {X 0,Y 476.218,Z 977.639,A -85,B 0,C 180,E1 13823.998,E2 13823.998} C_VEL
LIN {X 0,Y 496.439,Z 1030.939,A -85,B 0,C 180,E1 13826.512,E2 13826.512} C_VEL
LIN {X 0,Y 502.205,Z 1050.91,A -85,B 0,C 180,E1 13827.577,E2 13827.577} C_VEL
LIN {X 0,Y 498.339,Z 1091.029,A -85,B 0,C 180,E1 13829.413,E2 13829.413} C_VEL
LIN {X 0,Y 493.716,Z 1129.143,A -85,B 0,C 180,E1 13831.958,E2 13831.958} C_VEL
LIN {X 0,Y 489.082,Z 1162.63,A -85,B 0,C 180,E1 13835.02,E2 13835.02} C_VEL
LIN {X 0,Y 485.142,Z 1190.768,A -85,B 0,C 180,E1 13838.459,E2 13838.459} C_VEL
LIN {X 0,Y 481.981,Z 1214.812,A -85,B 0,C 180,E1 13842.375,E2 13842.375} C_VEL
LIN {X 0,Y 479.675,Z 1234.375,A -85,B 0,C 180,E1 13846.749,E2 13846.749} C_VEL
LIN {X 0,Y 478.553,Z 1248.244,A -85,B 0,C 180,E1 13851.338,E2 13851.338} C_VEL
LIN {X 0,Y 478.013,Z 1255.72,A -85,B 0,C 180,E1 13855.442,E2 13855.442} C_VEL
LIN {X 0,Y 478.014,Z 1258.951,A -85,B 0,C 180,E1 13859.987,E2 13859.987} C_VEL
LIN {X 0,Y 478.1,Z 1257.806,A -85,B 0,C 180,E1 13863.621,E2 13863.621} C_VEL
LIN {X 0,Y 478.668,Z 1251.671,A -85,B 0,C 180,E1 13868.176,E2 13868.176} C_VEL
LIN {X 0,Y 479.978,Z 1239.973,A -85,B 0,C 180,E1 13872.752,E2 13872.752} C_VEL
LIN {X 0,Y 482.364,Z 1223.366,A -85,B 0,C 180,E1 13877.037,E2 13877.037} C_VEL
LIN {X 0,Y 486.012,Z 1201.331,A -85,B 0,C 180,E1 13881.111,E2 13881.111} C_VEL
LIN {X 0,Y 490.551,Z 1174.901,A -85,B 0,C 180,E1 13884.742,E2 13884.742} C_VEL
LIN {X 0,Y 496.185,Z 1141.954,A -85,B 0,C 180,E1 13888.109,E2 13888.109} C_VEL
LIN {X 0,Y 501.857,Z 1104.944,A -85,B 0,C 180,E1 13890.864,E2 13890.864} C_VEL
LIN {X 0,Y 507.189,Z 1064.967,A -85,B 0,C 180,E1 13892.978,E2 13892.978} C_VEL
LIN {X 0,Y 508.23,Z 1048.468,A -85,B 0,C 180,E1 13893.729,E2 13893.729} C_VEL
LIN {X 0,Y 502.766,Z 1026.054,A -85,B 0,C 180,E1 13895.395,E2 13895.395} C_VEL
LIN {X 0,Y 494.201,Z 1007.091,A -85,B 0,C 180,E1 13897.501,E2 13897.501} C_VEL
LIN {X 0,Y 487.894,Z 996.528,A -85,B 0,C 180,E1 13899.405,E2 13899.405} C_VEL
LIN {X 0,Y 484.809,Z 991.3,A -85,B 0,C 180,E1 13900.709,E2 13900.709} C_VEL
LIN {X 0,Y 481.592,Z 985.05,A -85,B 0,C 180,E1 13903.223,E2 13903.223} C_VEL
LIN {X 0,Y 481.707,Z 985.725,A -85,B 0,C 180,E1 13906.267,E2 13906.267} C_VEL
LIN {X 0,Y 486.228,Z 993.406,A -85,B 0,C 180,E1 13909.17,E2 13909.17} C_VEL
LIN {X 0,Y 492.681,Z 1003.907,A -85,B 0,C 180,E1 13911.352,E2 13911.352} C_VEL
LIN {X 0,Y 497.786,Z 1015.111,A -85,B 0,C 180,E1 13912.756,E2 13912.756} C_VEL
LIN {X 0,Y 508.119,Z 1062.977,A -85,B 0,C 180,E1 13915.832,E2 13915.832} C_VEL
LIN {X 0,Y 502.904,Z 1106.903,A -85,B 0,C 180,E1 13917.452,E2 13917.452} C_VEL
LIN {X 0,Y 497.264,Z 1147.883,A -85,B 0,C 180,E1 13919.698,E2 13919.698} C_VEL
LIN {X 0,Y 491.666,Z 1185.646,A -85,B 0,C 180,E1 13922.575,E2 13922.575} C_VEL
LIN {X 0,Y 486.803,Z 1217.928,A -85,B 0,C 180,E1 13925.896,E2 13925.896} C_VEL
LIN {X 0,Y 482.775,Z 1246.465,A -85,B 0,C 180,E1 13929.812,E2 13929.812} C_VEL
LIN {X 0,Y 480.901,Z 1261.225,A -85,B 0,C 180,E1 13932.392,E2 13932.392} C_VEL
LIN {X 0,Y 475.988,Z 1270.075,A -85,B 0,C 180,E1 13934.115,E2 13934.115} C_VEL
LIN {X 0,Y 471.413,Z 1277.945,A -85,B 0,C 180,E1 13935.928,E2 13935.928} C_VEL
LIN {X 0,Y 470.471,Z 1291.658,A -85,B 0,C 180,E1 13940.274,E2 13940.274} C_VEL
LIN {X 0,Y 470.243,Z 1299.817,A -85,B 0,C 180,E1 13944.461,E2 13944.461} C_VEL
LIN {X 0,Y 470.184,Z 1303.275,A -85,B 0,C 180,E1 13948.162,E2 13948.162} C_VEL
LIN {X 0,Y 470.213,Z 1303.078,A -85,B 0,C 180,E1 13951.855,E2 13951.855} C_VEL
LIN {X 0,Y 470.3,Z 1297.842,A -85,B 0,C 180,E1 13956.483,E2 13956.483} C_VEL
LIN {X 0,Y 470.599,Z 1288.135,A -85,B 0,C 180,E1 13960.673,E2 13960.673} C_VEL
LIN {X 0,Y 471.691,Z 1273.128,A -85,B 0,C 180,E1 13964.9,E2 13964.9} C_VEL
LIN {X 0,Y 473.958,Z 1251.628,A -85,B 0,C 180,E1 13969.187,E2 13969.187} C_VEL
LIN {X 0,Y 477.442,Z 1225.158,A -85,B 0,C 180,E1 13973.068,E2 13973.068} C_VEL
LIN {X 0,Y 481.638,Z 1193.946,A -85,B 0,C 180,E1 13976.495,E2 13976.495} C_VEL
LIN {X 0,Y 486.367,Z 1158.479,A -85,B 0,C 180,E1 13979.375,E2 13979.375} C_VEL
LIN {X 0,Y 490.998,Z 1118.936,A -85,B 0,C 180,E1 13981.653,E2 13981.653} C_VEL
LIN {X 0,Y 496.839,Z 1064.567,A -85,B 0,C 180,E1 13983.794,E2 13983.794} C_VEL
LIN {X 0,Y 488.565,Z 1026.451,A -85,B 0,C 180,E1 13985.795,E2 13985.795} C_VEL
LIN {X 0,Y 476.966,Z 999.25,A -85,B 0,C 180,E1 13987.846,E2 13987.846} C_VEL
LIN {X 0,Y 472.691,Z 989.854,A -85,B 0,C 180,E1 13988.926,E2 13988.926} C_VEL
LIN {X 0,Y 468.235,Z 977.53,A -85,B 0,C 180,E1 13990.864,E2 13990.864} C_VEL
LIN {X 0,Y 468.186,Z 977.53,A -85,B 0,C 180,E1 13997.208,E2 13997.208} C_VEL
LIN {X 0,Y 468.169,Z 977.53,A -85,B 0,C 180,E1 14004.027,E2 14004.027} C_VEL
LIN {X 0,Y 468.336,Z 977.53,A -85,B 0,C 180,E1 14008.844,E2 14008.844} C_VEL
LIN {X 0,Y 468.606,Z 977.53,A -85,B 0,C 180,E1 14015.16,E2 14015.16} C_VEL
LIN {X 0,Y 468.833,Z 977.53,A -85,B 0,C 180,E1 14021.16,E2 14021.16} C_VEL
LIN {X 0,Y 468.922,Z 977.972,A -85,B 0,C 180,E1 14022.697,E2 14022.697} C_VEL
LIN {X 0,Y 483.545,Z 1008.076,A -85,B 0,C 180,E1 14026.074,E2 14026.074} C_VEL
LIN {X 0,Y 492.447,Z 1033.774,A -85,B 0,C 180,E1 14028.101,E2 14028.101} C_VEL
LIN {X 0,Y 487.856,Z 1086.861,A -85,B 0,C 180,E1 14030.065,E2 14030.065} C_VEL
LIN {X 0,Y 484.913,Z 1114.428,A -85,B 0,C 180,E1 14031.817,E2 14031.817} C_VEL
LIN {X 0,Y 481.422,Z 1138.807,A -85,B 0,C 180,E1 14034.142,E2 14034.142} C_VEL
LIN {X 0,Y 478.033,Z 1159.441,A -85,B 0,C 180,E1 14037.077,E2 14037.077} C_VEL
LIN {X 0,Y 475.161,Z 1175.204,A -85,B 0,C 180,E1 14040.47,E2 14040.47} C_VEL
LIN {X 0,Y 473.31,Z 1184.266,A -85,B 0,C 180,E1 14043.684,E2 14043.684} C_VEL
LIN {X 0,Y 471.991,Z 1188.959,A -85,B 0,C 180,E1 14047.39,E2 14047.39} C_VEL
LIN {X 0,Y 471.653,Z 1187.823,A -85,B 0,C 180,E1 14051.126,E2 14051.126} C_VEL
LIN {X 0,Y 472.026,Z 1180.646,A -85,B 0,C 180,E1 14054.893,E2 14054.893} C_VEL
LIN {X 0,Y 473.008,Z 1167.608,A -85,B 0,C 180,E1 14058.453,E2 14058.453} C_VEL
LIN {X 0,Y 474.458,Z 1149.359,A -85,B 0,C 180,E1 14061.637,E2 14061.637} C_VEL
LIN {X 0,Y 476.367,Z 1126.747,A -85,B 0,C 180,E1 14064.312,E2 14064.312} C_VEL
LIN {X 0,Y 478.362,Z 1100.377,A -85,B 0,C 180,E1 14066.435,E2 14066.435} C_VEL
LIN {X 0,Y 479.974,Z 1070.797,A -85,B 0,C 180,E1 14067.948,E2 14067.948} C_VEL
LIN {X 0,Y 480.856,Z 1021.756,A -85,B 0,C 180,E1 14069.278,E2 14069.278} C_VEL
LIN {X 0,Y 468.515,Z 977.53,A -85,B 0,C 180,E1 14070.992,E2 14070.992} C_VEL
LIN {X 0,Y 468.215,Z 977.53,A -85,B 0,C 180,E1 14077.955,E2 14077.955} C_VEL
LIN {X 0,Y 468.227,Z 977.53,A -85,B 0,C 180,E1 14084.593,E2 14084.593} C_VEL
LIN {X 0,Y 468.154,Z 977.53,A -85,B 0,C 180,E1 14090.981,E2 14090.981} C_VEL
LIN {X 0,Y 468.33,Z 977.53,A -85,B 0,C 180,E1 14097.283,E2 14097.283} C_VEL
LIN {X 0,Y 468.525,Z 977.53,A -85,B 0,C 180,E1 14103.068,E2 14103.068} C_VEL
LIN {X 0,Y 468.847,Z 977.53,A -85,B 0,C 180,E1 14109.614,E2 14109.614} C_VEL
LIN {X 0,Y 468.996,Z 977.53,A -85,B 0,C 180,E1 14115.784,E2 14115.784} C_VEL
LIN {X 0,Y 469.299,Z 977.53,A -85,B 0,C 180,E1 14120.701,E2 14120.701} C_VEL
LIN {X 0,Y 469.626,Z 977.53,A -85,B 0,C 180,E1 14126.291,E2 14126.291} C_VEL
LIN {X 0,Y 469.765,Z 977.53,A -85,B 0,C 180,E1 14131.84,E2 14131.84} C_VEL
LIN {X 0,Y 469.344,Z 977.53,A -85,B 0,C 180,E1 14137.411,E2 14137.411} C_VEL
LIN {X 0,Y 469.07,Z 977.53,A -85,B 0,C 180,E1 14143.06,E2 14143.06} C_VEL
LIN {X 0,Y 468.84,Z 977.53,A -85,B 0,C 180,E1 14148.847,E2 14148.847} C_VEL
LIN {X 0,Y 468.533,Z 977.53,A -85,B 0,C 180,E1 14155.088,E2 14155.088} C_VEL
LIN {X 0,Y 468.357,Z 977.53,A -85,B 0,C 180,E1 14161.164,E2 14161.164} C_VEL
LIN {X 0,Y 468.203,Z 977.53,A -85,B 0,C 180,E1 14167.934,E2 14167.934} C_VEL
LIN {X 0,Y 468.206,Z 977.53,A -85,B 0,C 180,E1 14174.591,E2 14174.591} C_VEL
LIN {X 0,Y 468.132,Z 977.53,A -85,B 0,C 180,E1 14180.958,E2 14180.958} C_VEL
LIN {X 0,Y 468.28,Z 977.53,A -85,B 0,C 180,E1 14183.471,E2 14183.471} C_VEL
LIN {X 0,Y 489.078,Z 1032.441,A -85,B 0,C 180,E1 14186.143,E2 14186.143} C_VEL
LIN {X 0,Y 494.894,Z 1052.988,A -85,B 0,C 180,E1 14187.26,E2 14187.26} C_VEL
LIN {X 0,Y 490.803,Z 1093.506,A -85,B 0,C 180,E1 14189.185,E2 14189.185} C_VEL
LIN {X 0,Y 486.127,Z 1130.694,A -85,B 0,C 180,E1 14191.734,E2 14191.734} C_VEL
LIN {X 0,Y 481.42,Z 1163.926,A -85,B 0,C 180,E1 14194.844,E2 14194.844} C_VEL
LIN {X 0,Y 477.166,Z 1193.53,A -85,B 0,C 180,E1 14198.57,E2 14198.57} C_VEL
LIN {X 0,Y 473.843,Z 1218.141,A -85,B 0,C 180,E1 14202.783,E2 14202.783} C_VEL
LIN {X 0,Y 471.697,Z 1236.002,A -85,B 0,C 180,E1 14206.993,E2 14206.993} C_VEL
LIN {X 0,Y 470.597,Z 1249.424,A -85,B 0,C 180,E1 14211.657,E2 14211.657} C_VEL
LIN {X 0,Y 470.119,Z 1257.055,A -85,B 0,C 180,E1 14216.291,E2 14216.291} C_VEL
LIN {X 0,Y 470.123,Z 1259.333,A -85,B 0,C 180,E1 14219.987,E2 14219.987} C_VEL
LIN {X 0,Y 470.242,Z 1258.28,A -85,B 0,C 180,E1 14223.681,E2 14223.681} C_VEL
LIN {X 0,Y 470.845,Z 1252.234,A -85,B 0,C 180,E1 14228.312,E2 14228.312} C_VEL
LIN {X 0,Y 472.234,Z 1240.63,A -85,B 0,C 180,E1 14232.965,E2 14232.965} C_VEL
LIN {X 0,Y 474.856,Z 1223.785,A -85,B 0,C 180,E1 14237.391,E2 14237.391} C_VEL
LIN {X 0,Y 478.764,Z 1201.483,A -85,B 0,C 180,E1 14241.575,E2 14241.575} C_VEL
LIN {X 0,Y 483.644,Z 1174.966,A -85,B 0,C 180,E1 14245.259,E2 14245.259} C_VEL
LIN {X 0,Y 489.585,Z 1142.201,A -85,B 0,C 180,E1 14248.649,E2 14248.649} C_VEL
LIN {X 0,Y 495.581,Z 1105.44,A -85,B 0,C 180,E1 14251.427,E2 14251.427} C_VEL
LIN {X 0,Y 501.324,Z 1065.204,A -85,B 0,C 180,E1 14253.591,E2 14253.591} C_VEL
LIN {X 0,Y 502.411,Z 1051.467,A -85,B 0,C 180,E1 14254.234,E2 14254.234} C_VEL
LIN {X 0,Y 497.638,Z 1030.376,A -85,B 0,C 180,E1 14255.889,E2 14255.889} C_VEL
LIN {X 0,Y 490.215,Z 1012.778,A -85,B 0,C 180,E1 14257.952,E2 14257.952} C_VEL
LIN {X 0,Y 484.341,Z 1002.427,A -85,B 0,C 180,E1 14259.937,E2 14259.937} C_VEL
LIN {X 0,Y 481.896,Z 998.269,A -85,B 0,C 180,E1 14261.093,E2 14261.093} C_VEL
LIN {X 0,Y 479.426,Z 992.629,A -85,B 0,C 180,E1 14263.382,E2 14263.382} C_VEL
LIN {X 0,Y 479.51,Z 993.408,A -85,B 0,C 180,E1 14266.145,E2 14266.145} C_VEL
LIN {X 0,Y 483.534,Z 1000.824,A -85,B 0,C 180,E1 14268.955,E2 14268.955} C_VEL
LIN {X 0,Y 489.49,Z 1011.159,A -85,B 0,C 180,E1 14271.11,E2 14271.11} C_VEL
LIN {X 0,Y 493.418,Z 1020.403,A -85,B 0,C 180,E1 14272.286,E2 14272.286} C_VEL
LIN {X 0,Y 502.069,Z 1064.965,A -85,B 0,C 180,E1 14275.274,E2 14275.274} C_VEL
LIN {X 0,Y 496.393,Z 1108.84,A -85,B 0,C 180,E1 14276.976,E2 14276.976} C_VEL
LIN {X 0,Y 490.238,Z 1150.41,A -85,B 0,C 180,E1 14279.346,E2 14279.346} C_VEL
LIN {X 0,Y 484.212,Z 1188.322,A -85,B 0,C 180,E1 14282.371,E2 14282.371} C_VEL
LIN {X 0,Y 479.15,Z 1219.772,A -85,B 0,C 180,E1 14285.735,E2 14285.735} C_VEL
LIN {X 0,Y 475.031,Z 1247.505,A -85,B 0,C 180,E1 14289.675,E2 14289.675} C_VEL
LIN {X 0,Y 472.284,Z 1269.295,A -85,B 0,C 180,E1 14293.836,E2 14293.836} C_VEL
LIN {X 0,Y 471.413,Z 1277.945,A -85,B 0,C 180,E1 14295.928,E2 14295.928} C_VEL
LIN {X 0,Y 466.933,Z 1284.762,A -85,B 0,C 180,E1 14297.825,E2 14297.825} C_VEL
LIN {X 0,Y 462.668,Z 1290.564,A -85,B 0,C 180,E1 14299.802,E2 14299.802} C_VEL
LIN {X 0,Y 462.345,Z 1299.486,A -85,B 0,C 180,E1 14304.366,E2 14304.366} C_VEL
LIN {X 0,Y 462.297,Z 1302.886,A -85,B 0,C 180,E1 14308.13,E2 14308.13} C_VEL
LIN {X 0,Y 462.325,Z 1302.643,A -85,B 0,C 180,E1 14311.887,E2 14311.887} C_VEL
LIN {X 0,Y 462.404,Z 1297.303,A -85,B 0,C 180,E1 14316.595,E2 14316.595} C_VEL
LIN {X 0,Y 462.766,Z 1287.331,A -85,B 0,C 180,E1 14320.9,E2 14320.9} C_VEL
LIN {X 0,Y 463.92,Z 1272.281,A -85,B 0,C 180,E1 14325.156,E2 14325.156} C_VEL
LIN {X 0,Y 466.128,Z 1251.791,A -85,B 0,C 180,E1 14329.304,E2 14329.304} C_VEL
LIN {X 0,Y 469.77,Z 1224.863,A -85,B 0,C 180,E1 14333.32,E2 14333.32} C_VEL
LIN {X 0,Y 474.185,Z 1193.173,A -85,B 0,C 180,E1 14336.841,E2 14336.841} C_VEL
LIN {X 0,Y 479.199,Z 1156.753,A -85,B 0,C 180,E1 14339.812,E2 14339.812} C_VEL
LIN {X 0,Y 483.774,Z 1118.181,A -85,B 0,C 180,E1 14342.05,E2 14342.05} C_VEL
LIN {X 0,Y 489.442,Z 1073.43,A -85,B 0,C 180,E1 14344.037,E2 14344.037} C_VEL
LIN {X 0,Y 489.834,Z 1062.115,A -85,B 0,C 180,E1 14344.484,E2 14344.484} C_VEL
LIN {X 0,Y 481.959,Z 1027.368,A -85,B 0,C 180,E1 14346.454,E2 14346.454} C_VEL
LIN {X 0,Y 470.417,Z 1000.78,A -85,B 0,C 180,E1 14348.641,E2 14348.641} C_VEL
LIN {X 0,Y 464.686,Z 989.084,A -85,B 0,C 180,E1 14350.023,E2 14350.023} C_VEL
LIN {X 0,Y 460.34,Z 977.53,A -85,B 0,C 180,E1 14352.069,E2 14352.069} C_VEL
LIN {X 0,Y 460.278,Z 977.53,A -85,B 0,C 180,E1 14358.845,E2 14358.845} C_VEL
LIN {X 0,Y 460.254,Z 977.53,A -85,B 0,C 180,E1 14365.407,E2 14365.407} C_VEL
LIN {X 0,Y 460.471,Z 977.53,A -85,B 0,C 180,E1 14370.442,E2 14370.442} C_VEL
LIN {X 0,Y 460.826,Z 977.53,A -85,B 0,C 180,E1 14377.048,E2 14377.048} C_VEL
LIN {X 0,Y 460.932,Z 977.64,A -85,B 0,C 180,E1 14381.415,E2 14381.415} C_VEL
LIN {X 0,Y 463.472,Z 983.278,A -85,B 0,C 180,E1 14382.149,E2 14382.149} C_VEL
LIN {X 0,Y 475.609,Z 1006.992,A -85,B 0,C 180,E1 14385.102,E2 14385.102} C_VEL
LIN {X 0,Y 485.544,Z 1033.91,A -85,B 0,C 180,E1 14387.47,E2 14387.47} C_VEL
LIN {X 0,Y 480.957,Z 1089.828,A -85,B 0,C 180,E1 14389.692,E2 14389.692} C_VEL
LIN {X 0,Y 477.688,Z 1117.948,A -85,B 0,C 180,E1 14391.578,E2 14391.578} C_VEL
LIN {X 0,Y 473.923,Z 1142.264,A -85,B 0,C 180,E1 14394.049,E2 14394.049} C_VEL
LIN {X 0,Y 470.461,Z 1161.815,A -85,B 0,C 180,E1 14396.965,E2 14396.965} C_VEL
LIN {X 0,Y 467.417,Z 1177.217,A -85,B 0,C 180,E1 14400.478,E2 14400.478} C_VEL
LIN {X 0,Y 465.481,Z 1185.853,A -85,B 0,C 180,E1 14403.746,E2 14403.746} C_VEL
LIN {X 0,Y 464.136,Z 1190.11,A -85,B 0,C 180,E1 14407.516,E2 14407.516} C_VEL
LIN {X 0,Y 463.82,Z 1188.387,A -85,B 0,C 180,E1 14411.413,E2 14411.413} C_VEL
LIN {X 0,Y 464.23,Z 1180.899,A -85,B 0,C 180,E1 14415.149,E2 14415.149} C_VEL
LIN {X 0,Y 465.282,Z 1167.319,A -85,B 0,C 180,E1 14418.771,E2 14418.771} C_VEL
LIN {X 0,Y 466.768,Z 1149.051,A -85,B 0,C 180,E1 14421.928,E2 14421.928} C_VEL
LIN {X 0,Y 468.867,Z 1125.099,A -85,B 0,C 180,E1 14424.727,E2 14424.727} C_VEL
LIN {X 0,Y 470.974,Z 1097.689,A -85,B 0,C 180,E1 14426.874,E2 14426.874} C_VEL
LIN {X 0,Y 472.524,Z 1067.357,A -85,B 0,C 180,E1 14428.356,E2 14428.356} C_VEL
LIN {X 0,Y 473.276,Z 1022.853,A -85,B 0,C 180,E1 14429.552,E2 14429.552} C_VEL
LIN {X 0,Y 460.55,Z 977.53,A -85,B 0,C 180,E1 14431.362,E2 14431.362} C_VEL
LIN {X 0,Y 460.297,Z 977.53,A -85,B 0,C 180,E1 14437.794,E2 14437.794} C_VEL
LIN {X 0,Y 460.277,Z 977.53,A -85,B 0,C 180,E1 14443.748,E2 14443.748} C_VEL
LIN {X 0,Y 460.259,Z 977.53,A -85,B 0,C 180,E1 14449.231,E2 14449.231} C_VEL
LIN {X 0,Y 460.296,Z 977.53,A -85,B 0,C 180,E1 14455.959,E2 14455.959} C_VEL
LIN {X 0,Y 460.57,Z 977.53,A -85,B 0,C 180,E1 14462.565,E2 14462.565} C_VEL
LIN {X 0,Y 460.849,Z 977.53,A -85,B 0,C 180,E1 14468.787,E2 14468.787} C_VEL
LIN {X 0,Y 461.058,Z 977.53,A -85,B 0,C 180,E1 14474.748,E2 14474.748} C_VEL
LIN {X 0,Y 461.367,Z 977.53,A -85,B 0,C 180,E1 14480.54,E2 14480.54} C_VEL
LIN {X 0,Y 461.714,Z 977.53,A -85,B 0,C 180,E1 14486.228,E2 14486.228} C_VEL
LIN {X 0,Y 461.857,Z 977.53,A -85,B 0,C 180,E1 14491.871,E2 14491.871} C_VEL
LIN {X 0,Y 461.421,Z 977.53,A -85,B 0,C 180,E1 14497.539,E2 14497.539} C_VEL
LIN {X 0,Y 461.147,Z 977.53,A -85,B 0,C 180,E1 14503.289,E2 14503.289} C_VEL
LIN {X 0,Y 460.912,Z 977.53,A -85,B 0,C 180,E1 14509.184,E2 14509.184} C_VEL
LIN {X 0,Y 460.606,Z 977.53,A -85,B 0,C 180,E1 14515.31,E2 14515.31} C_VEL
LIN {X 0,Y 460.441,Z 977.53,A -85,B 0,C 180,E1 14521.762,E2 14521.762} C_VEL
LIN {X 0,Y 460.284,Z 977.53,A -85,B 0,C 180,E1 14528.706,E2 14528.706} C_VEL
LIN {X 0,Y 460.26,Z 977.53,A -85,B 0,C 180,E1 14533.726,E2 14533.726} C_VEL
LIN {X 0,Y 460.227,Z 977.53,A -85,B 0,C 180,E1 14539.21,E2 14539.21} C_VEL
LIN {X 0,Y 460.343,Z 977.53,A -85,B 0,C 180,E1 14542.932,E2 14542.932} C_VEL
LIN {X 0,Y 481.335,Z 1032.953,A -85,B 0,C 180,E1 14545.712,E2 14545.712} C_VEL
LIN {X 0,Y 487.605,Z 1055.011,A -85,B 0,C 180,E1 14546.94,E2 14546.94} C_VEL
LIN {X 0,Y 483.467,Z 1094.181,A -85,B 0,C 180,E1 14548.849,E2 14548.849} C_VEL
LIN {X 0,Y 478.739,Z 1130.864,A -85,B 0,C 180,E1 14551.4,E2 14551.4} C_VEL
LIN {X 0,Y 473.897,Z 1164.066,A -85,B 0,C 180,E1 14554.543,E2 14554.543} C_VEL
LIN {X 0,Y 469.611,Z 1192.948,A -85,B 0,C 180,E1 14558.207,E2 14558.207} C_VEL
LIN {X 0,Y 466.142,Z 1217.908,A -85,B 0,C 180,E1 14562.489,E2 14562.489} C_VEL
LIN {X 0,Y 463.908,Z 1235.979,A -85,B 0,C 180,E1 14566.771,E2 14566.771} C_VEL
LIN {X 0,Y 462.735,Z 1249.576,A -85,B 0,C 180,E1 14571.514,E2 14571.514} C_VEL
LIN {X 0,Y 462.227,Z 1257.352,A -85,B 0,C 180,E1 14576.228,E2 14576.228} C_VEL
LIN {X 0,Y 462.236,Z 1259.715,A -85,B 0,C 180,E1 14579.987,E2 14579.987} C_VEL
LIN {X 0,Y 462.359,Z 1258.765,A -85,B 0,C 180,E1 14583.744,E2 14583.744} C_VEL
LIN {X 0,Y 463.008,Z 1252.818,A -85,B 0,C 180,E1 14588.454,E2 14588.454} C_VEL
LIN {X 0,Y 464.514,Z 1241.322,A -85,B 0,C 180,E1 14593.184,E2 14593.184} C_VEL
LIN {X 0,Y 467.301,Z 1224.602,A -85,B 0,C 180,E1 14597.681,E2 14597.681} C_VEL
LIN {X 0,Y 471.425,Z 1202.507,A -85,B 0,C 180,E1 14601.923,E2 14601.923} C_VEL
LIN {X 0,Y 476.592,Z 1176.26,A -85,B 0,C 180,E1 14605.652,E2 14605.652} C_VEL
LIN {X 0,Y 482.829,Z 1143.881,A -85,B 0,C 180,E1 14609.088,E2 14609.088} C_VEL
LIN {X 0,Y 489.409,Z 1106.22,A -85,B 0,C 180,E1 14612,E2 14612} C_VEL
LIN {X 0,Y 495.776,Z 1064.783,A -85,B 0,C 180,E1 14614.265,E2 14614.265} C_VEL
LIN {X 0,Y 496.547,Z 1053.199,A -85,B 0,C 180,E1 14614.852,E2 14614.852} C_VEL
LIN {X 0,Y 492.277,Z 1033.324,A -85,B 0,C 180,E1 14616.533,E2 14616.533} C_VEL
LIN {X 0,Y 485.466,Z 1016.422,A -85,B 0,C 180,E1 14618.724,E2 14618.724} C_VEL
LIN {X 0,Y 479.765,Z 1005.881,A -85,B 0,C 180,E1 14621.131,E2 14621.131} C_VEL
LIN {X 0,Y 477.304,Z 1000.238,A -85,B 0,C 180,E1 14623.492,E2 14623.492} C_VEL
LIN {X 0,Y 477.349,Z 1001.171,A -85,B 0,C 180,E1 14626.063,E2 14626.063} C_VEL
LIN {X 0,Y 480.929,Z 1008.21,A -85,B 0,C 180,E1 14628.757,E2 14628.757} C_VEL
LIN {X 0,Y 486.379,Z 1018.292,A -85,B 0,C 180,E1 14630.864,E2 14630.864} C_VEL
LIN {X 0,Y 489.198,Z 1026.255,A -85,B 0,C 180,E1 14631.832,E2 14631.832} C_VEL
LIN {X 0,Y 496.186,Z 1067.436,A -85,B 0,C 180,E1 14634.723,E2 14634.723} C_VEL
LIN {X 0,Y 490.141,Z 1109.95,A -85,B 0,C 180,E1 14636.435,E2 14636.435} C_VEL
LIN {X 0,Y 483.527,Z 1151.377,A -85,B 0,C 180,E1 14638.874,E2 14638.874} C_VEL
LIN {X 0,Y 477.139,Z 1188.91,A -85,B 0,C 180,E1 14641.949,E2 14641.949} C_VEL
LIN {X 0,Y 471.682,Z 1220.885,A -85,B 0,C 180,E1 14645.467,E2 14645.467} C_VEL
LIN {X 0,Y 467.373,Z 1248.123,A -85,B 0,C 180,E1 14649.453,E2 14649.453} C_VEL
LIN {X 0,Y 464.367,Z 1270.996,A -85,B 0,C 180,E1 14653.99,E2 14653.99} C_VEL
LIN {X 0,Y 462.82,Z 1287.541,A -85,B 0,C 180,E1 14658.68,E2 14658.68} C_VEL
LIN {X 0,Y 462.668,Z 1290.564,A -85,B 0,C 180,E1 14659.802,E2 14659.802} C_VEL
LIN {X 0,Y 460.013,Z 1294.216,A -85,B 0,C 180,E1 14661.333,E2 14661.333} C_VEL
LIN {X 0,Y 454.563,Z 1298.307,A -85,B 0,C 180,E1 14663.676,E2 14663.676} C_VEL
LIN {X 0,Y 454.465,Z 1298.701,A -85,B 0,C 180,E1 14663.949,E2 14663.949} C_VEL
LIN {X 0,Y 454.404,Z 1302.497,A -85,B 0,C 180,E1 14668.098,E2 14668.098} C_VEL
LIN {X 0,Y 454.449,Z 1302.201,A -85,B 0,C 180,E1 14671.92,E2 14671.92} C_VEL
LIN {X 0,Y 454.52,Z 1296.747,A -85,B 0,C 180,E1 14676.71,E2 14676.71} C_VEL
LIN {X 0,Y 454.858,Z 1287.253,A -85,B 0,C 180,E1 14680.877,E2 14680.877} C_VEL
LIN {X 0,Y 456.094,Z 1271.382,A -85,B 0,C 180,E1 14685.422,E2 14685.422} C_VEL
LIN {X 0,Y 458.434,Z 1250.655,A -85,B 0,C 180,E1 14689.641,E2 14689.641} C_VEL
LIN {X 0,Y 462.095,Z 1224.419,A -85,B 0,C 180,E1 14693.596,E2 14693.596} C_VEL
LIN {X 0,Y 466.507,Z 1193.806,A -85,B 0,C 180,E1 14697.058,E2 14697.058} C_VEL
LIN {X 0,Y 471.638,Z 1157.72,A -85,B 0,C 180,E1 14700.075,E2 14700.075} C_VEL
LIN {X 0,Y 479.316,Z 1102.423,A -85,B 0,C 180,E1 14703.36,E2 14703.36} C_VEL
LIN {X 0,Y 483.382,Z 1064.613,A -85,B 0,C 180,E1 14704.956,E2 14704.956} C_VEL
LIN {X 0,Y 476.456,Z 1031.273,A -85,B 0,C 180,E1 14706.945,E2 14706.945} C_VEL
LIN {X 0,Y 465.062,Z 1004.495,A -85,B 0,C 180,E1 14709.25,E2 14709.25} C_VEL
LIN {X 0,Y 456.141,Z 987.277,A -85,B 0,C 180,E1 14711.441,E2 14711.441} C_VEL
LIN {X 0,Y 452.378,Z 977.53,A -85,B 0,C 180,E1 14713.298,E2 14713.298} C_VEL
LIN {X 0,Y 452.284,Z 977.53,A -85,B 0,C 180,E1 14720.418,E2 14720.418} C_VEL
LIN {X 0,Y 452.344,Z 977.53,A -85,B 0,C 180,E1 14726.888,E2 14726.888} C_VEL
LIN {X 0,Y 452.59,Z 977.53,A -85,B 0,C 180,E1 14732.068,E2 14732.068} C_VEL
LIN {X 0,Y 452.91,Z 977.53,A -85,B 0,C 180,E1 14738.424,E2 14738.424} C_VEL
LIN {X 0,Y 452.95,Z 978.28,A -85,B 0,C 180,E1 14740.01,E2 14740.01} C_VEL
LIN {X 0,Y 456.093,Z 983.755,A -85,B 0,C 180,E1 14740.934,E2 14740.934} C_VEL
LIN {X 0,Y 467.88,Z 1006.504,A -85,B 0,C 180,E1 14744.09,E2 14744.09} C_VEL
LIN {X 0,Y 477.769,Z 1031.763,A -85,B 0,C 180,E1 14746.579,E2 14746.579} C_VEL
LIN {X 0,Y 479.41,Z 1040.147,A -85,B 0,C 180,E1 14747.149,E2 14747.149} C_VEL
LIN {X 0,Y 474.44,Z 1089.84,A -85,B 0,C 180,E1 14749.142,E2 14749.142} C_VEL
LIN {X 0,Y 471.06,Z 1117.401,A -85,B 0,C 180,E1 14750.992,E2 14750.992} C_VEL
LIN {X 0,Y 467.003,Z 1142.218,A -85,B 0,C 180,E1 14753.493,E2 14753.493} C_VEL
LIN {X 0,Y 463.144,Z 1162.74,A -85,B 0,C 180,E1 14756.589,E2 14756.589} C_VEL
LIN {X 0,Y 460.042,Z 1177.673,A -85,B 0,C 180,E1 14760.013,E2 14760.013} C_VEL
LIN {X 0,Y 457.679,Z 1187.435,A -85,B 0,C 180,E1 14763.81,E2 14763.81} C_VEL
LIN {X 0,Y 456.288,Z 1191.188,A -85,B 0,C 180,E1 14767.646,E2 14767.646} C_VEL
LIN {X 0,Y 455.998,Z 1189.176,A -85,B 0,C 180,E1 14771.513,E2 14771.513} C_VEL
LIN {X 0,Y 456.355,Z 1182.451,A -85,B 0,C 180,E1 14774.924,E2 14774.924} C_VEL
LIN {X 0,Y 457.352,Z 1169.286,A -85,B 0,C 180,E1 14778.608,E2 14778.608} C_VEL
LIN {X 0,Y 458.931,Z 1150.823,A -85,B 0,C 180,E1 14781.919,E2 14781.919} C_VEL
LIN {X 0,Y 460.912,Z 1128.314,A -85,B 0,C 180,E1 14784.664,E2 14784.664} C_VEL
LIN {X 0,Y 463.06,Z 1101.648,A -85,B 0,C 180,E1 14786.883,E2 14786.883} C_VEL
LIN {X 0,Y 464.76,Z 1072.833,A -85,B 0,C 180,E1 14788.419,E2 14788.419} C_VEL
LIN {X 0,Y 465.735,Z 1024.376,A -85,B 0,C 180,E1 14789.82,E2 14789.82} C_VEL
LIN {X 0,Y 452.649,Z 977.53,A -85,B 0,C 180,E1 14791.697,E2 14791.697} C_VEL
LIN {X 0,Y 452.399,Z 977.53,A -85,B 0,C 180,E1 14797.089,E2 14797.089} C_VEL
LIN {X 0,Y 452.286,Z 977.53,A -85,B 0,C 180,E1 14802.506,E2 14802.506} C_VEL
LIN {X 0,Y 452.26,Z 977.53,A -85,B 0,C 180,E1 14807.914,E2 14807.914} C_VEL
LIN {X 0,Y 452.361,Z 977.53,A -85,B 0,C 180,E1 14813.52,E2 14813.52} C_VEL
LIN {X 0,Y 452.564,Z 977.53,A -85,B 0,C 180,E1 14820.536,E2 14820.536} C_VEL
LIN {X 0,Y 452.785,Z 977.53,A -85,B 0,C 180,E1 14826.313,E2 14826.313} C_VEL
LIN {X 0,Y 453.052,Z 977.53,A -85,B 0,C 180,E1 14832.472,E2 14832.472} C_VEL
LIN {X 0,Y 453.301,Z 977.53,A -85,B 0,C 180,E1 14838.421,E2 14838.421} C_VEL
LIN {X 0,Y 453.721,Z 977.53,A -85,B 0,C 180,E1 14844.241,E2 14844.241} C_VEL
LIN {X 0,Y 454.007,Z 977.53,A -85,B 0,C 180,E1 14849.991,E2 14849.991} C_VEL
LIN {X 0,Y 453.705,Z 977.53,A -85,B 0,C 180,E1 14855.741,E2 14855.741} C_VEL
LIN {X 0,Y 453.291,Z 977.53,A -85,B 0,C 180,E1 14861.561,E2 14861.561} C_VEL
LIN {X 0,Y 453.046,Z 977.53,A -85,B 0,C 180,E1 14867.509,E2 14867.509} C_VEL
LIN {X 0,Y 452.744,Z 977.53,A -85,B 0,C 180,E1 14873.67,E2 14873.67} C_VEL
LIN {X 0,Y 452.558,Z 977.53,A -85,B 0,C 180,E1 14880.137,E2 14880.137} C_VEL
LIN {X 0,Y 452.379,Z 977.53,A -85,B 0,C 180,E1 14887.068,E2 14887.068} C_VEL
LIN {X 0,Y 452.281,Z 977.53,A -85,B 0,C 180,E1 14892.506,E2 14892.506} C_VEL
LIN {X 0,Y 452.234,Z 977.53,A -85,B 0,C 180,E1 14897.911,E2 14897.911} C_VEL
LIN {X 0,Y 452.408,Z 978.165,A -85,B 0,C 180,E1 14902.447,E2 14902.447} C_VEL
LIN {X 0,Y 473.285,Z 1032.447,A -85,B 0,C 180,E1 14905.212,E2 14905.212} C_VEL
LIN {X 0,Y 480.299,Z 1056.615,A -85,B 0,C 180,E1 14906.603,E2 14906.603} C_VEL
LIN {X 0,Y 476.007,Z 1095.911,A -85,B 0,C 180,E1 14908.572,E2 14908.572} C_VEL
LIN {X 0,Y 471.196,Z 1132.12,A -85,B 0,C 180,E1 14911.149,E2 14911.149} C_VEL
LIN {X 0,Y 466.218,Z 1165.261,A -85,B 0,C 180,E1 14914.351,E2 14914.351} C_VEL
LIN {X 0,Y 461.84,Z 1193.983,A -85,B 0,C 180,E1 14918.075,E2 14918.075} C_VEL
LIN {X 0,Y 458.302,Z 1218.764,A -85,B 0,C 180,E1 14922.428,E2 14922.428} C_VEL
LIN {X 0,Y 455.934,Z 1237.539,A -85,B 0,C 180,E1 14927.024,E2 14927.024} C_VEL
LIN {X 0,Y 454.842,Z 1250.242,A -85,B 0,C 180,E1 14931.615,E2 14931.615} C_VEL
LIN {X 0,Y 454.338,Z 1257.641,A -85,B 0,C 180,E1 14936.162,E2 14936.162} C_VEL
LIN {X 0,Y 454.349,Z 1260.096,A -85,B 0,C 180,E1 14939.986,E2 14939.986} C_VEL
LIN {X 0,Y 454.495,Z 1259.26,A -85,B 0,C 180,E1 14943.809,E2 14943.809} C_VEL
LIN {X 0,Y 455.203,Z 1253.424,A -85,B 0,C 180,E1 14948.6,E2 14948.6} C_VEL
LIN {X 0,Y 456.789,Z 1242.052,A -85,B 0,C 180,E1 14953.411,E2 14953.411} C_VEL
LIN {X 0,Y 459.968,Z 1224.414,A -85,B 0,C 180,E1 14958.221,E2 14958.221} C_VEL
LIN {X 0,Y 464.43,Z 1202.152,A -85,B 0,C 180,E1 14962.525,E2 14962.525} C_VEL
LIN {X 0,Y 470.433,Z 1173.916,A -85,B 0,C 180,E1 14966.527,E2 14966.527} C_VEL
LIN {X 0,Y 477.125,Z 1140.684,A -85,B 0,C 180,E1 14969.994,E2 14969.994} C_VEL
LIN {X 0,Y 483.973,Z 1103.965,A -85,B 0,C 180,E1 14972.803,E2 14972.803} C_VEL
LIN {X 0,Y 490.568,Z 1063.306,A -85,B 0,C 180,E1 14975.018,E2 14975.018} C_VEL
LIN {X 0,Y 490.8,Z 1053.967,A -85,B 0,C 180,E1 14975.577,E2 14975.577} C_VEL
LIN {X 0,Y 486.581,Z 1034.904,A -85,B 0,C 180,E1 14977.394,E2 14977.394} C_VEL
LIN {X 0,Y 480.964,Z 1020.802,A -85,B 0,C 180,E1 14979.514,E2 14979.514} C_VEL
LIN {X 0,Y 476.917,Z 1012.836,A -85,B 0,C 180,E1 14981.541,E2 14981.541} C_VEL
LIN {X 0,Y 475.093,Z 1007.821,A -85,B 0,C 180,E1 14983.741,E2 14983.741} C_VEL
LIN {X 0,Y 475.199,Z 1008.836,A -85,B 0,C 180,E1 14985.963,E2 14985.963} C_VEL
LIN {X 0,Y 478.263,Z 1015.415,A -85,B 0,C 180,E1 14988.508,E2 14988.508} C_VEL
LIN {X 0,Y 483.559,Z 1025.931,A -85,B 0,C 180,E1 14990.702,E2 14990.702} C_VEL
LIN {X 0,Y 485.321,Z 1033.563,A -85,B 0,C 180,E1 14991.481,E2 14991.481} C_VEL
LIN {X 0,Y 490.323,Z 1070.381,A -85,B 0,C 180,E1 14994.149,E2 14994.149} C_VEL
LIN {X 0,Y 483.485,Z 1114.258,A -85,B 0,C 180,E1 14996.022,E2 14996.022} C_VEL
LIN {X 0,Y 476.347,Z 1155.583,A -85,B 0,C 180,E1 14998.618,E2 14998.618} C_VEL
LIN {X 0,Y 469.934,Z 1190.626,A -85,B 0,C 180,E1 15001.611,E2 15001.611} C_VEL
LIN {X 0,Y 464.007,Z 1223.304,A -85,B 0,C 180,E1 15005.345,E2 15005.345} C_VEL
LIN {X 0,Y 459.315,Z 1251.142,A -85,B 0,C 180,E1 15009.64,E2 15009.64} C_VEL
LIN {X 0,Y 456.466,Z 1271.974,A -85,B 0,C 180,E1 15014.006,E2 15014.006} C_VEL
LIN {X 0,Y 454.949,Z 1287.273,A -85,B 0,C 180,E1 15018.482,E2 15018.482} C_VEL
LIN {X 0,Y 454.506,Z 1297.769,A -85,B 0,C 180,E1 15023.308,E2 15023.308} C_VEL
LIN {X 0,Y 454.465,Z 1298.701,A -85,B 0,C 180,E1 15023.949,E2 15023.949} C_VEL
LIN {X 0,Y 451.936,Z 1300.663,A -85,B 0,C 180,E1 15025.555,E2 15025.555} C_VEL
LIN {X 0,Y 446.598,Z 1302.089,A -85,B 0,C 180,E1 15027.988,E2 15027.988} C_VEL
LIN {X 0,Y 446.498,Z 1302.135,A -85,B 0,C 180,E1 15028.27,E2 15028.27} C_VEL
LIN {X 0,Y 446.554,Z 1301.752,A -85,B 0,C 180,E1 15031.954,E2 15031.954} C_VEL
LIN {X 0,Y 446.642,Z 1296.183,A -85,B 0,C 180,E1 15036.828,E2 15036.828} C_VEL
LIN {X 0,Y 446.999,Z 1286.516,A -85,B 0,C 180,E1 15041.078,E2 15041.078} C_VEL
LIN {X 0,Y 448.295,Z 1270.467,A -85,B 0,C 180,E1 15045.698,E2 15045.698} C_VEL
LIN {X 0,Y 450.703,Z 1250.081,A -85,B 0,C 180,E1 15049.885,E2 15049.885} C_VEL
LIN {X 0,Y 454.406,Z 1224.075,A -85,B 0,C 180,E1 15053.858,E2 15053.858} C_VEL
LIN {X 0,Y 459.072,Z 1193.002,A -85,B 0,C 180,E1 15057.414,E2 15057.414} C_VEL
LIN {X 0,Y 464.423,Z 1156.331,A -85,B 0,C 180,E1 15060.502,E2 15060.502} C_VEL
LIN {X 0,Y 471.514,Z 1110.871,A -85,B 0,C 180,E1 15063.468,E2 15063.468} C_VEL
LIN {X 0,Y 476.995,Z 1066.473,A -85,B 0,C 180,E1 15065.482,E2 15065.482} C_VEL
LIN {X 0,Y 470.723,Z 1034.439,A -85,B 0,C 180,E1 15067.494,E2 15067.494} C_VEL
LIN {X 0,Y 459.761,Z 1008.074,A -85,B 0,C 180,E1 15069.904,E2 15069.904} C_VEL
LIN {X 0,Y 448.174,Z 987.033,A -85,B 0,C 180,E1 15072.806,E2 15072.806} C_VEL
LIN {X 0,Y 444.369,Z 977.53,A -85,B 0,C 180,E1 15074.876,E2 15074.876} C_VEL
LIN {X 0,Y 444.322,Z 977.53,A -85,B 0,C 180,E1 15081.677,E2 15081.677} C_VEL
LIN {X 0,Y 444.471,Z 977.53,A -85,B 0,C 180,E1 15086.965,E2 15086.965} C_VEL
LIN {X 0,Y 444.704,Z 977.53,A -85,B 0,C 180,E1 15093.726,E2 15093.726} C_VEL
LIN {X 0,Y 445.024,Z 978.035,A -85,B 0,C 180,E1 15098.308,E2 15098.308} C_VEL
LIN {X 0,Y 447.694,Z 983.437,A -85,B 0,C 180,E1 15099.294,E2 15099.294} C_VEL
LIN {X 0,Y 456.844,Z 999.461,A -85,B 0,C 180,E1 15102.052,E2 15102.052} C_VEL
LIN {X 0,Y 467.355,Z 1022.316,A -85,B 0,C 180,E1 15104.893,E2 15104.893} C_VEL
LIN {X 0,Y 473.284,Z 1041.011,A -85,B 0,C 180,E1 15106.561,E2 15106.561} C_VEL
LIN {X 0,Y 467.865,Z 1091.02,A -85,B 0,C 180,E1 15108.632,E2 15108.632} C_VEL
LIN {X 0,Y 464.294,Z 1118.419,A -85,B 0,C 180,E1 15110.505,E2 15110.505} C_VEL
LIN {X 0,Y 459.815,Z 1144.002,A -85,B 0,C 180,E1 15113.154,E2 15113.154} C_VEL
LIN {X 0,Y 455.869,Z 1163.723,A -85,B 0,C 180,E1 15116.202,E2 15116.202} C_VEL
LIN {X 0,Y 452.689,Z 1178.179,A -85,B 0,C 180,E1 15119.534,E2 15119.534} C_VEL
LIN {X 0,Y 450.347,Z 1187.251,A -85,B 0,C 180,E1 15122.906,E2 15122.906} C_VEL
LIN {X 0,Y 449.011,Z 1191.317,A -85,B 0,C 180,E1 15125.824,E2 15125.824} C_VEL
LIN {X 0,Y 448.175,Z 1191.779,A -85,B 0,C 180,E1 15129.745,E2 15129.745} C_VEL
LIN {X 0,Y 448.322,Z 1186.3,A -85,B 0,C 180,E1 15133.698,E2 15133.698} C_VEL
LIN {X 0,Y 448.966,Z 1176.225,A -85,B 0,C 180,E1 15137.189,E2 15137.189} C_VEL
LIN {X 0,Y 450.354,Z 1160.006,A -85,B 0,C 180,E1 15140.7,E2 15140.7} C_VEL
LIN {X 0,Y 452.445,Z 1138.207,A -85,B 0,C 180,E1 15143.835,E2 15143.835} C_VEL
LIN {X 0,Y 454.617,Z 1112.505,A -85,B 0,C 180,E1 15146.353,E2 15146.353} C_VEL
LIN {X 0,Y 456.678,Z 1083.19,A -85,B 0,C 180,E1 15148.23,E2 15148.23} C_VEL
LIN {X 0,Y 457.916,Z 1051.985,A -85,B 0,C 180,E1 15149.38,E2 15149.38} C_VEL
LIN {X 0,Y 458.177,Z 1025.715,A -85,B 0,C 180,E1 15150.088,E2 15150.088} C_VEL
LIN {X 0,Y 444.664,Z 977.53,A -85,B 0,C 180,E1 15152.097,E2 15152.097} C_VEL
LIN {X 0,Y 444.392,Z 977.53,A -85,B 0,C 180,E1 15158.335,E2 15158.335} C_VEL
LIN {X 0,Y 444.315,Z 977.53,A -85,B 0,C 180,E1 15164.248,E2 15164.248} C_VEL
LIN {X 0,Y 444.309,Z 977.53,A -85,B 0,C 180,E1 15169.599,E2 15169.599} C_VEL
LIN {X 0,Y 444.493,Z 977.53,A -85,B 0,C 180,E1 15176.935,E2 15176.935} C_VEL
LIN {X 0,Y 444.708,Z 977.53,A -85,B 0,C 180,E1 15183.698,E2 15183.698} C_VEL
LIN {X 0,Y 445.042,Z 977.53,A -85,B 0,C 180,E1 15190.085,E2 15190.085} C_VEL
LIN {X 0,Y 445.284,Z 977.53,A -85,B 0,C 180,E1 15196.21,E2 15196.21} C_VEL
LIN {X 0,Y 445.63,Z 977.53,A -85,B 0,C 180,E1 15202.174,E2 15202.174} C_VEL
LIN {X 0,Y 445.991,Z 977.53,A -85,B 0,C 180,E1 15208.044,E2 15208.044} C_VEL
LIN {X 0,Y 445.889,Z 977.53,A -85,B 0,C 180,E1 15213.888,E2 15213.888} C_VEL
LIN {X 0,Y 445.502,Z 977.53,A -85,B 0,C 180,E1 15219.782,E2 15219.782} C_VEL
LIN {X 0,Y 445.179,Z 977.53,A -85,B 0,C 180,E1 15225.792,E2 15225.792} C_VEL
LIN {X 0,Y 444.909,Z 977.53,A -85,B 0,C 180,E1 15231.992,E2 15231.992} C_VEL
LIN {X 0,Y 444.63,Z 977.53,A -85,B 0,C 180,E1 15238.486,E2 15238.486} C_VEL
LIN {X 0,Y 444.463,Z 977.53,A -85,B 0,C 180,E1 15245.409,E2 15245.409} C_VEL
LIN {X 0,Y 444.326,Z 977.53,A -85,B 0,C 180,E1 15251.374,E2 15251.374} C_VEL
LIN {X 0,Y 444.287,Z 977.53,A -85,B 0,C 180,E1 15256.978,E2 15256.978} C_VEL
LIN {X 0,Y 444.459,Z 978.206,A -85,B 0,C 180,E1 15261.898,E2 15261.898} C_VEL
LIN {X 0,Y 465.198,Z 1031.964,A -85,B 0,C 180,E1 15264.706,E2 15264.706} C_VEL
LIN {X 0,Y 473.024,Z 1058.176,A -85,B 0,C 180,E1 15266.262,E2 15266.262} C_VEL
LIN {X 0,Y 468.544,Z 1097.539,A -85,B 0,C 180,E1 15268.285,E2 15268.285} C_VEL
LIN {X 0,Y 463.595,Z 1133.708,A -85,B 0,C 180,E1 15270.925,E2 15270.925} C_VEL
LIN {X 0,Y 458.389,Z 1167.451,A -85,B 0,C 180,E1 15274.275,E2 15274.275} C_VEL
LIN {X 0,Y 453.837,Z 1196.508,A -85,B 0,C 180,E1 15278.184,E2 15278.184} C_VEL
LIN {X 0,Y 450.44,Z 1219.603,A -85,B 0,C 180,E1 15282.364,E2 15282.364} C_VEL
LIN {X 0,Y 448.154,Z 1237.473,A -85,B 0,C 180,E1 15286.795,E2 15286.795} C_VEL
LIN {X 0,Y 446.939,Z 1250.862,A -85,B 0,C 180,E1 15291.702,E2 15291.702} C_VEL
LIN {X 0,Y 446.446,Z 1257.924,A -85,B 0,C 180,E1 15296.094,E2 15296.094} C_VEL
LIN {X 0,Y 446.458,Z 1260.476,A -85,B 0,C 180,E1 15299.986,E2 15299.986} C_VEL
LIN {X 0,Y 446.614,Z 1259.756,A -85,B 0,C 180,E1 15303.876,E2 15303.876} C_VEL
LIN {X 0,Y 447.389,Z 1254.047,A -85,B 0,C 180,E1 15308.752,E2 15308.752} C_VEL
LIN {X 0,Y 449.083,Z 1242.82,A -85,B 0,C 180,E1 15313.646,E2 15313.646} C_VEL
LIN {X 0,Y 452.492,Z 1225.35,A -85,B 0,C 180,E1 15318.533,E2 15318.533} C_VEL
LIN {X 0,Y 457.21,Z 1203.319,A -85,B 0,C 180,E1 15322.9,E2 15322.9} C_VEL
LIN {X 0,Y 463.504,Z 1175.431,A -85,B 0,C 180,E1 15326.956,E2 15326.956} C_VEL
LIN {X 0,Y 470.818,Z 1141.57,A -85,B 0,C 180,E1 15330.572,E2 15330.572} C_VEL
LIN {X 0,Y 478.047,Z 1105.439,A -85,B 0,C 180,E1 15333.397,E2 15333.397} C_VEL
LIN {X 0,Y 485.297,Z 1064.271,A -85,B 0,C 180,E1 15335.698,E2 15335.698} C_VEL
LIN {X 0,Y 485.075,Z 1053.133,A -85,B 0,C 180,E1 15336.493,E2 15336.493} C_VEL
LIN {X 0,Y 480.812,Z 1035.351,A -85,B 0,C 180,E1 15338.501,E2 15338.501} C_VEL
LIN {X 0,Y 476.185,Z 1023.913,A -85,B 0,C 180,E1 15340.663,E2 15340.663} C_VEL
LIN {X 0,Y 473.789,Z 1019.062,A -85,B 0,C 180,E1 15342.282,E2 15342.282} C_VEL
LIN {X 0,Y 472.93,Z 1015.408,A -85,B 0,C 180,E1 15343.992,E2 15343.992} C_VEL
LIN {X 0,Y 473.049,Z 1016.432,A -85,B 0,C 180,E1 15345.843,E2 15345.843} C_VEL
LIN {X 0,Y 475.844,Z 1023.086,A -85,B 0,C 180,E1 15348.381,E2 15348.381} C_VEL
LIN {X 0,Y 480.654,Z 1033.647,A -85,B 0,C 180,E1 15350.521,E2 15350.521} C_VEL
LIN {X 0,Y 484.767,Z 1072.542,A -85,B 0,C 180,E1 15353.518,E2 15353.518} C_VEL
LIN {X 0,Y 477.199,Z 1116.761,A -85,B 0,C 180,E1 15355.508,E2 15355.508} C_VEL
LIN {X 0,Y 469.728,Z 1156.96,A -85,B 0,C 180,E1 15358.124,E2 15358.124} C_VEL
LIN {X 0,Y 462.59,Z 1193.669,A -85,B 0,C 180,E1 15361.386,E2 15361.386} C_VEL
LIN {X 0,Y 456.312,Z 1225.665,A -85,B 0,C 180,E1 15365.223,E2 15365.223} C_VEL
LIN {X 0,Y 451.537,Z 1252.524,A -85,B 0,C 180,E1 15369.546,E2 15369.546} C_VEL
LIN {X 0,Y 448.584,Z 1272.896,A -85,B 0,C 180,E1 15373.997,E2 15373.997} C_VEL
LIN {X 0,Y 447.098,Z 1287.03,A -85,B 0,C 180,E1 15378.277,E2 15378.277} C_VEL
LIN {X 0,Y 446.626,Z 1297.45,A -85,B 0,C 180,E1 15383.189,E2 15383.189} C_VEL
LIN {X 0,Y 446.508,Z 1302.106,A -85,B 0,C 180,E1 15388.064,E2 15388.064} C_VEL
LIN {X 0,Y 446.498,Z 1302.135,A -85,B 0,C 180,E1 15388.27,E2 15388.27} C_VEL
LIN {X 0,Y 443.992,Z 1302.285,A -85,B 0,C 180,E1 15389.924,E2 15389.924} C_VEL
LIN {X 0,Y 438.608,Z 1300.751,A -85,B 0,C 180,E1 15392.69,E2 15392.69} C_VEL
LIN {X 0,Y 438.759,Z 1295.599,A -85,B 0,C 180,E1 15396.952,E2 15396.952} C_VEL
LIN {X 0,Y 439.149,Z 1285.449,A -85,B 0,C 180,E1 15401.39,E2 15401.39} C_VEL
LIN {X 0,Y 440.605,Z 1268.464,A -85,B 0,C 180,E1 15406.235,E2 15406.235} C_VEL
LIN {X 0,Y 443.386,Z 1245.891,A -85,B 0,C 180,E1 15410.776,E2 15410.776} C_VEL
LIN {X 0,Y 447.61,Z 1217.774,A -85,B 0,C 180,E1 15414.91,E2 15414.91} C_VEL
LIN {X 0,Y 452.586,Z 1186.098,A -85,B 0,C 180,E1 15418.369,E2 15418.369} C_VEL
LIN {X 0,Y 460.873,Z 1135.721,A -85,B 0,C 180,E1 15422.487,E2 15422.487} C_VEL
LIN {X 0,Y 467.509,Z 1094.959,A -85,B 0,C 180,E1 15424.848,E2 15424.848} C_VEL
LIN {X 0,Y 470.722,Z 1068.796,A -85,B 0,C 180,E1 15426.002,E2 15426.002} C_VEL
LIN {X 0,Y 465.203,Z 1038.094,A -85,B 0,C 180,E1 15428.031,E2 15428.031} C_VEL
LIN {X 0,Y 455.152,Z 1012.998,A -85,B 0,C 180,E1 15430.429,E2 15430.429} C_VEL
LIN {X 0,Y 444.306,Z 992.768,A -85,B 0,C 180,E1 15433.329,E2 15433.329} C_VEL
LIN {X 0,Y 437.841,Z 982.029,A -85,B 0,C 180,E1 15435.58,E2 15435.58} C_VEL
LIN {X 0,Y 436.405,Z 977.53,A -85,B 0,C 180,E1 15436.829,E2 15436.829} C_VEL
LIN {X 0,Y 436.399,Z 977.53,A -85,B 0,C 180,E1 15443.846,E2 15443.846} C_VEL
LIN {X 0,Y 436.657,Z 977.53,A -85,B 0,C 180,E1 15450.954,E2 15450.954} C_VEL
LIN {X 0,Y 436.991,Z 978.105,A -85,B 0,C 180,E1 15456.233,E2 15456.233} C_VEL
LIN {X 0,Y 439.876,Z 983.618,A -85,B 0,C 180,E1 15457.491,E2 15457.491} C_VEL
LIN {X 0,Y 442.271,Z 987.648,A -85,B 0,C 180,E1 15458.399,E2 15458.399} C_VEL
LIN {X 0,Y 448.603,Z 998.039,A -85,B 0,C 180,E1 15460.508,E2 15460.508} C_VEL
LIN {X 0,Y 458.474,Z 1018.225,A -85,B 0,C 180,E1 15463.457,E2 15463.457} C_VEL
LIN {X 0,Y 466.955,Z 1042.148,A -85,B 0,C 180,E1 15465.914,E2 15465.914} C_VEL
LIN {X 0,Y 461.126,Z 1094.54,A -85,B 0,C 180,E1 15468.224,E2 15468.224} C_VEL
LIN {X 0,Y 456.94,Z 1123.415,A -85,B 0,C 180,E1 15470.35,E2 15470.35} C_VEL
LIN {X 0,Y 452.315,Z 1147.565,A -85,B 0,C 180,E1 15473.04,E2 15473.04} C_VEL
LIN {X 0,Y 448.236,Z 1166.521,A -85,B 0,C 180,E1 15476.138,E2 15476.138} C_VEL
LIN {X 0,Y 444.914,Z 1180.26,A -85,B 0,C 180,E1 15479.526,E2 15479.526} C_VEL
LIN {X 0,Y 442.515,Z 1188.871,A -85,B 0,C 180,E1 15482.958,E2 15482.958} C_VEL
LIN {X 0,Y 441.166,Z 1192.608,A -85,B 0,C 180,E1 15485.928,E2 15485.928} C_VEL
LIN {X 0,Y 440.338,Z 1192.58,A -85,B 0,C 180,E1 15489.921,E2 15489.921} C_VEL
LIN {X 0,Y 440.501,Z 1186.649,A -85,B 0,C 180,E1 15493.946,E2 15493.946} C_VEL
LIN {X 0,Y 441.287,Z 1175.134,A -85,B 0,C 180,E1 15497.755,E2 15497.755} C_VEL
LIN {X 0,Y 442.797,Z 1157.776,A -85,B 0,C 180,E1 15501.333,E2 15501.333} C_VEL
LIN {X 0,Y 445.017,Z 1135.884,A -85,B 0,C 180,E1 15504.369,E2 15504.369} C_VEL
LIN {X 0,Y 447.221,Z 1110.036,A -85,B 0,C 180,E1 15506.823,E2 15506.823} C_VEL
LIN {X 0,Y 449.196,Z 1081.588,A -85,B 0,C 180,E1 15508.592,E2 15508.592} C_VEL
LIN {X 0,Y 450.513,Z 1047.064,A -85,B 0,C 180,E1 15509.805,E2 15509.805} C_VEL
LIN {X 0,Y 450.558,Z 1026.872,A -85,B 0,C 180,E1 15510.374,E2 15510.374} C_VEL
LIN {X 0,Y 436.712,Z 977.53,A -85,B 0,C 180,E1 15512.541,E2 15512.541} C_VEL
LIN {X 0,Y 436.453,Z 977.53,A -85,B 0,C 180,E1 15518.689,E2 15518.689} C_VEL
LIN {X 0,Y 436.426,Z 977.53,A -85,B 0,C 180,E1 15523.992,E2 15523.992} C_VEL
LIN {X 0,Y 436.384,Z 977.53,A -85,B 0,C 180,E1 15529.824,E2 15529.824} C_VEL
LIN {X 0,Y 436.546,Z 977.53,A -85,B 0,C 180,E1 15536.428,E2 15536.428} C_VEL
LIN {X 0,Y 436.762,Z 977.53,A -85,B 0,C 180,E1 15543.181,E2 15543.181} C_VEL
LIN {X 0,Y 437.08,Z 977.53,A -85,B 0,C 180,E1 15549.706,E2 15549.706} C_VEL
LIN {X 0,Y 437.372,Z 977.53,A -85,B 0,C 180,E1 15555.974,E2 15555.974} C_VEL
LIN {X 0,Y 437.709,Z 977.53,A -85,B 0,C 180,E1 15562.031,E2 15562.031} C_VEL
LIN {X 0,Y 438.096,Z 977.53,A -85,B 0,C 180,E1 15568.009,E2 15568.009} C_VEL
LIN {X 0,Y 437.994,Z 977.53,A -85,B 0,C 180,E1 15573.958,E2 15573.958} C_VEL
LIN {X 0,Y 437.566,Z 977.53,A -85,B 0,C 180,E1 15579.961,E2 15579.961} C_VEL
LIN {X 0,Y 437.242,Z 977.53,A -85,B 0,C 180,E1 15586.086,E2 15586.086} C_VEL
LIN {X 0,Y 436.959,Z 977.53,A -85,B 0,C 180,E1 15592.414,E2 15592.414} C_VEL
LIN {X 0,Y 436.647,Z 977.53,A -85,B 0,C 180,E1 15599.056,E2 15599.056} C_VEL
LIN {X 0,Y 436.538,Z 977.53,A -85,B 0,C 180,E1 15603.725,E2 15603.725} C_VEL
LIN {X 0,Y 436.422,Z 977.53,A -85,B 0,C 180,E1 15610.182,E2 15610.182} C_VEL
LIN {X 0,Y 436.393,Z 977.53,A -85,B 0,C 180,E1 15616.803,E2 15616.803} C_VEL
LIN {X 0,Y 436.476,Z 977.53,A -85,B 0,C 180,E1 15621.313,E2 15621.313} C_VEL
LIN {X 0,Y 457.724,Z 1033.12,A -85,B 0,C 180,E1 15624.285,E2 15624.285} C_VEL
LIN {X 0,Y 465.726,Z 1059.922,A -85,B 0,C 180,E1 15625.926,E2 15625.926} C_VEL
LIN {X 0,Y 461.107,Z 1099.063,A -85,B 0,C 180,E1 15627.99,E2 15627.99} C_VEL
LIN {X 0,Y 455.863,Z 1136.089,A -85,B 0,C 180,E1 15630.766,E2 15630.766} C_VEL
LIN {X 0,Y 450.387,Z 1170.594,A -85,B 0,C 180,E1 15634.327,E2 15634.327} C_VEL
LIN {X 0,Y 445.772,Z 1199.307,A -85,B 0,C 180,E1 15638.355,E2 15638.355} C_VEL
LIN {X 0,Y 442.288,Z 1222.662,A -85,B 0,C 180,E1 15642.793,E2 15642.793} C_VEL
LIN {X 0,Y 439.981,Z 1240.625,A -85,B 0,C 180,E1 15647.557,E2 15647.557} C_VEL
LIN {X 0,Y 438.973,Z 1252.004,A -85,B 0,C 180,E1 15652.05,E2 15652.05} C_VEL
LIN {X 0,Y 438.56,Z 1258.202,A -85,B 0,C 180,E1 15656.024,E2 15656.024} C_VEL
LIN {X 0,Y 438.568,Z 1260.859,A -85,B 0,C 180,E1 15659.986,E2 15659.986} C_VEL
LIN {X 0,Y 438.758,Z 1260.239,A -85,B 0,C 180,E1 15663.946,E2 15663.946} C_VEL
LIN {X 0,Y 439.564,Z 1254.672,A -85,B 0,C 180,E1 15668.909,E2 15668.909} C_VEL
LIN {X 0,Y 441.392,Z 1243.622,A -85,B 0,C 180,E1 15673.888,E2 15673.888} C_VEL
LIN {X 0,Y 445.021,Z 1226.353,A -85,B 0,C 180,E1 15678.856,E2 15678.856} C_VEL
LIN {X 0,Y 450.007,Z 1204.583,A -85,B 0,C 180,E1 15683.288,E2 15683.288} C_VEL
LIN {X 0,Y 456.629,Z 1177.08,A -85,B 0,C 180,E1 15687.396,E2 15687.396} C_VEL
LIN {X 0,Y 464.332,Z 1143.976,A -85,B 0,C 180,E1 15691.045,E2 15691.045} C_VEL
LIN {X 0,Y 472.235,Z 1107.265,A -85,B 0,C 180,E1 15694.002,E2 15694.002} C_VEL
LIN {X 0,Y 480.141,Z 1066.089,A -85,B 0,C 180,E1 15696.374,E2 15696.374} C_VEL
LIN {X 0,Y 479.79,Z 1054.708,A -85,B 0,C 180,E1 15697.296,E2 15697.296} C_VEL
LIN {X 0,Y 476.043,Z 1038.075,A -85,B 0,C 180,E1 15699.423,E2 15699.423} C_VEL
LIN {X 0,Y 472.208,Z 1027.655,A -85,B 0,C 180,E1 15701.848,E2 15701.848} C_VEL
LIN {X 0,Y 470.81,Z 1023.019,A -85,B 0,C 180,E1 15704.24,E2 15704.24} C_VEL
LIN {X 0,Y 470.948,Z 1024.334,A -85,B 0,C 180,E1 15705.854,E2 15705.854} C_VEL
LIN {X 0,Y 473.339,Z 1030.443,A -85,B 0,C 180,E1 15708.178,E2 15708.178} C_VEL
LIN {X 0,Y 476.851,Z 1039.626,A -85,B 0,C 180,E1 15710.033,E2 15710.033} C_VEL
LIN {X 0,Y 479.498,Z 1074.319,A -85,B 0,C 180,E1 15712.844,E2 15712.844} C_VEL
LIN {X 0,Y 471.252,Z 1118.331,A -85,B 0,C 180,E1 15714.908,E2 15714.908} C_VEL
LIN {X 0,Y 462.889,Z 1160.06,A -85,B 0,C 180,E1 15717.735,E2 15717.735} C_VEL
LIN {X 0,Y 455.205,Z 1196.597,A -85,B 0,C 180,E1 15721.15,E2 15721.15} C_VEL
LIN {X 0,Y 449.077,Z 1225.969,A -85,B 0,C 180,E1 15724.797,E2 15724.797} C_VEL
LIN {X 0,Y 444.183,Z 1251.716,A -85,B 0,C 180,E1 15729.021,E2 15729.021} C_VEL
LIN {X 0,Y 440.905,Z 1272.146,A -85,B 0,C 180,E1 15733.539,E2 15733.539} C_VEL
LIN {X 0,Y 439.244,Z 1286.808,A -85,B 0,C 180,E1 15738.064,E2 15738.064} C_VEL
LIN {X 0,Y 438.741,Z 1297.149,A -85,B 0,C 180,E1 15743.066,E2 15743.066} C_VEL
LIN {X 0,Y 438.612,Z 1301.717,A -85,B 0,C 180,E1 15748.029,E2 15748.029} C_VEL
LIN {X 0,Y 438.68,Z 1301.298,A -85,B 0,C 180,E1 15751.989,E2 15751.989} C_VEL
LIN {X 0,Y 438.608,Z 1300.751,A -85,B 0,C 180,E1 15752.69,E2 15752.69} C_VEL
LIN {X 0,Y 436.132,Z 1299.167,A -85,B 0,C 180,E1 15754.366,E2 15754.366} C_VEL
LIN {X 0,Y 430.876,Z 1294.88,A -85,B 0,C 180,E1 15757.142,E2 15757.142} C_VEL
LIN {X 0,Y 431.411,Z 1283.072,A -85,B 0,C 180,E1 15762.175,E2 15762.175} C_VEL
LIN {X 0,Y 433.082,Z 1265.291,A -85,B 0,C 180,E1 15767.049,E2 15767.049} C_VEL
LIN {X 0,Y 436.288,Z 1241.51,A -85,B 0,C 180,E1 15771.665,E2 15771.665} C_VEL
LIN {X 0,Y 440.597,Z 1214.039,A -85,B 0,C 180,E1 15775.607,E2 15775.607} C_VEL
LIN {X 0,Y 445.785,Z 1181.306,A -85,B 0,C 180,E1 15779.121,E2 15779.121} C_VEL
LIN {X 0,Y 452.684,Z 1144.497,A -85,B 0,C 180,E1 15782.393,E2 15782.393} C_VEL
LIN {X 0,Y 459.722,Z 1104.723,A -85,B 0,C 180,E1 15784.948,E2 15784.948} C_VEL
LIN {X 0,Y 464.437,Z 1070.71,A -85,B 0,C 180,E1 15786.567,E2 15786.567} C_VEL
LIN {X 0,Y 459.756,Z 1041.932,A -85,B 0,C 180,E1 15788.562,E2 15788.562} C_VEL
LIN {X 0,Y 450.595,Z 1017.902,A -85,B 0,C 180,E1 15790.982,E2 15790.982} C_VEL
LIN {X 0,Y 440.703,Z 998.779,A -85,B 0,C 180,E1 15793.804,E2 15793.804} C_VEL
LIN {X 0,Y 433.861,Z 987.525,A -85,B 0,C 180,E1 15796.266,E2 15796.266} C_VEL
LIN {X 0,Y 431.243,Z 983.557,A -85,B 0,C 180,E1 15797.416,E2 15797.416} C_VEL
LIN {X 0,Y 428.579,Z 978.585,A -85,B 0,C 180,E1 15798.868,E2 15798.868} C_VEL
LIN {X 0,Y 428.484,Z 977.53,A -85,B 0,C 180,E1 15799.712,E2 15799.712} C_VEL
LIN {X 0,Y 428.484,Z 977.53,A -85,B 0,C 180,E1 15805.563,E2 15805.563} C_VEL
LIN {X 0,Y 428.779,Z 977.53,A -85,B 0,C 180,E1 15812.671,E2 15812.671} C_VEL
LIN {X 0,Y 428.917,Z 978.377,A -85,B 0,C 180,E1 15813.467,E2 15813.467} C_VEL
LIN {X 0,Y 432.065,Z 983.783,A -85,B 0,C 180,E1 15815.236,E2 15815.236} C_VEL
LIN {X 0,Y 433.947,Z 986.295,A -85,B 0,C 180,E1 15816.079,E2 15816.079} C_VEL
LIN {X 0,Y 441.228,Z 998.079,A -85,B 0,C 180,E1 15818.986,E2 15818.986} C_VEL
LIN {X 0,Y 451.558,Z 1018.838,A -85,B 0,C 180,E1 15822.438,E2 15822.438} C_VEL
LIN {X 0,Y 459.954,Z 1041.812,A -85,B 0,C 180,E1 15825.06,E2 15825.06} C_VEL
LIN {X 0,Y 460.829,Z 1047.042,A -85,B 0,C 180,E1 15825.468,E2 15825.468} C_VEL
LIN {X 0,Y 454.777,Z 1095.094,A -85,B 0,C 180,E1 15827.63,E2 15827.63} C_VEL
LIN {X 0,Y 450.686,Z 1122.007,A -85,B 0,C 180,E1 15829.604,E2 15829.604} C_VEL
LIN {X 0,Y 445.96,Z 1145.99,A -85,B 0,C 180,E1 15832.204,E2 15832.204} C_VEL
LIN {X 0,Y 441.302,Z 1166.237,A -85,B 0,C 180,E1 15835.466,E2 15835.466} C_VEL
LIN {X 0,Y 437.615,Z 1180.852,A -85,B 0,C 180,E1 15839.022,E2 15839.022} C_VEL
LIN {X 0,Y 434.706,Z 1190.486,A -85,B 0,C 180,E1 15843.011,E2 15843.011} C_VEL
LIN {X 0,Y 433.326,Z 1193.871,A -85,B 0,C 180,E1 15846.035,E2 15846.035} C_VEL
LIN {X 0,Y 432.498,Z 1193.339,A -85,B 0,C 180,E1 15850.102,E2 15850.102} C_VEL
LIN {X 0,Y 432.686,Z 1186.979,A -85,B 0,C 180,E1 15854.203,E2 15854.203} C_VEL
LIN {X 0,Y 433.551,Z 1174.899,A -85,B 0,C 180,E1 15858.083,E2 15858.083} C_VEL
LIN {X 0,Y 435.016,Z 1158.482,A -85,B 0,C 180,E1 15861.466,E2 15861.466} C_VEL
LIN {X 0,Y 437.309,Z 1136.257,A -85,B 0,C 180,E1 15864.582,E2 15864.582} C_VEL
LIN {X 0,Y 439.557,Z 1110.634,A -85,B 0,C 180,E1 15867.052,E2 15867.052} C_VEL
LIN {X 0,Y 441.689,Z 1080.828,A -85,B 0,C 180,E1 15868.92,E2 15868.92} C_VEL
LIN {X 0,Y 443.028,Z 1045.731,A -85,B 0,C 180,E1 15870.148,E2 15870.148} C_VEL
LIN {X 0,Y 443.046,Z 1028.279,A -85,B 0,C 180,E1 15870.658,E2 15870.658} C_VEL
LIN {X 0,Y 428.786,Z 977.53,A -85,B 0,C 180,E1 15872.835,E2 15872.835} C_VEL
LIN {X 0,Y 428.537,Z 977.53,A -85,B 0,C 180,E1 15879.542,E2 15879.542} C_VEL
LIN {X 0,Y 428.467,Z 977.53,A -85,B 0,C 180,E1 15885.029,E2 15885.029} C_VEL
LIN {X 0,Y 428.476,Z 977.53,A -85,B 0,C 180,E1 15891.093,E2 15891.093} C_VEL
LIN {X 0,Y 428.67,Z 977.53,A -85,B 0,C 180,E1 15898.049,E2 15898.049} C_VEL
LIN {X 0,Y 428.922,Z 977.53,A -85,B 0,C 180,E1 15904.907,E2 15904.907} C_VEL
LIN {X 0,Y 429.217,Z 977.53,A -85,B 0,C 180,E1 15911.465,E2 15911.465} C_VEL
LIN {X 0,Y 429.509,Z 977.53,A -85,B 0,C 180,E1 15917.77,E2 15917.77} C_VEL
LIN {X 0,Y 429.949,Z 977.53,A -85,B 0,C 180,E1 15923.921,E2 15923.921} C_VEL
LIN {X 0,Y 430.328,Z 977.53,A -85,B 0,C 180,E1 15929.991,E2 15929.991} C_VEL
LIN {X 0,Y 429.928,Z 977.53,A -85,B 0,C 180,E1 15936.06,E2 15936.06} C_VEL
LIN {X 0,Y 429.501,Z 977.53,A -85,B 0,C 180,E1 15942.211,E2 15942.211} C_VEL
LIN {X 0,Y 429.194,Z 977.53,A -85,B 0,C 180,E1 15948.517,E2 15948.517} C_VEL
LIN {X 0,Y 428.88,Z 977.53,A -85,B 0,C 180,E1 15955.075,E2 15955.075} C_VEL
LIN {X 0,Y 428.657,Z 977.53,A -85,B 0,C 180,E1 15962.01,E2 15962.01} C_VEL
LIN {X 0,Y 428.529,Z 977.53,A -85,B 0,C 180,E1 15968.916,E2 15968.916} C_VEL
LIN {X 0,Y 428.446,Z 977.53,A -85,B 0,C 180,E1 15975.005,E2 15975.005} C_VEL
LIN {X 0,Y 428.514,Z 977.53,A -85,B 0,C 180,E1 15980.716,E2 15980.716} C_VEL
LIN {X 0,Y 450.209,Z 1034.361,A -85,B 0,C 180,E1 15983.863,E2 15983.863} C_VEL
LIN {X 0,Y 458.407,Z 1061.751,A -85,B 0,C 180,E1 15985.585,E2 15985.585} C_VEL
LIN {X 0,Y 453.693,Z 1100.515,A -85,B 0,C 180,E1 15987.687,E2 15987.687} C_VEL
LIN {X 0,Y 448.098,Z 1138.657,A -85,B 0,C 180,E1 15990.626,E2 15990.626} C_VEL
LIN {X 0,Y 442.708,Z 1171.486,A -85,B 0,C 180,E1 15994.114,E2 15994.114} C_VEL
LIN {X 0,Y 438.057,Z 1199.737,A -85,B 0,C 180,E1 15998.147,E2 15998.147} C_VEL
LIN {X 0,Y 434.572,Z 1222.329,A -85,B 0,C 180,E1 16002.485,E2 16002.485} C_VEL
LIN {X 0,Y 432.17,Z 1240.512,A -85,B 0,C 180,E1 16007.329,E2 16007.329} C_VEL
LIN {X 0,Y 431.11,Z 1252.103,A -85,B 0,C 180,E1 16011.904,E2 16011.904} C_VEL
LIN {X 0,Y 430.67,Z 1258.472,A -85,B 0,C 180,E1 16015.951,E2 16015.951} C_VEL
LIN {X 0,Y 430.677,Z 1261.24,A -85,B 0,C 180,E1 16019.986,E2 16019.986} C_VEL
LIN {X 0,Y 430.876,Z 1260.724,A -85,B 0,C 180,E1 16024.018,E2 16024.018} C_VEL
LIN {X 0,Y 431.775,Z 1255.305,A -85,B 0,C 180,E1 16029.071,E2 16029.071} C_VEL
LIN {X 0,Y 433.717,Z 1244.443,A -85,B 0,C 180,E1 16034.139,E2 16034.139} C_VEL
LIN {X 0,Y 437.581,Z 1227.42,A -85,B 0,C 180,E1 16039.189,E2 16039.189} C_VEL
LIN {X 0,Y 442.85,Z 1205.941,A -85,B 0,C 180,E1 16043.688,E2 16043.688} C_VEL
LIN {X 0,Y 449.819,Z 1178.865,A -85,B 0,C 180,E1 16047.846,E2 16047.846} C_VEL
LIN {X 0,Y 458.204,Z 1145.338,A -85,B 0,C 180,E1 16051.647,E2 16051.647} C_VEL
LIN {X 0,Y 466.877,Z 1107.866,A -85,B 0,C 180,E1 16054.729,E2 16054.729} C_VEL
LIN {X 0,Y 475.494,Z 1063.908,A -85,B 0,C 180,E1 16057.366,E2 16057.366} C_VEL
LIN {X 0,Y 473.415,Z 1048.366,A -85,B 0,C 180,E1 16059.184,E2 16059.184} C_VEL
LIN {X 0,Y 470.501,Z 1037.756,A -85,B 0,C 180,E1 16061.26,E2 16061.26} C_VEL
LIN {X 0,Y 468.746,Z 1030.706,A -85,B 0,C 180,E1 16064.002,E2 16064.002} C_VEL
LIN {X 0,Y 468.736,Z 1031.642,A -85,B 0,C 180,E1 16065.605,E2 16065.605} C_VEL
LIN {X 0,Y 470.778,Z 1037.925,A -85,B 0,C 180,E1 16068.015,E2 16068.015} C_VEL
LIN {X 0,Y 473.166,Z 1045.519,A -85,B 0,C 180,E1 16069.517,E2 16069.517} C_VEL
LIN {X 0,Y 474.099,Z 1077.771,A -85,B 0,C 180,E1 16072.211,E2 16072.211} C_VEL
LIN {X 0,Y 465.462,Z 1120.09,A -85,B 0,C 180,E1 16074.289,E2 16074.289} C_VEL
LIN {X 0,Y 456.389,Z 1161.723,A -85,B 0,C 180,E1 16077.218,E2 16077.218} C_VEL
LIN {X 0,Y 448.314,Z 1197.475,A -85,B 0,C 180,E1 16080.664,E2 16080.664} C_VEL
LIN {X 0,Y 441.498,Z 1228.097,A -85,B 0,C 180,E1 16084.605,E2 16084.605} C_VEL
LIN {X 0,Y 436.203,Z 1254.455,A -85,B 0,C 180,E1 16089.152,E2 16089.152} C_VEL
LIN {X 0,Y 432.747,Z 1275.584,A -85,B 0,C 180,E1 16094.196,E2 16094.196} C_VEL
LIN {X 0,Y 431.225,Z 1289.208,A -85,B 0,C 180,E1 16098.867,E2 16098.867} C_VEL
LIN {X 0,Y 430.778,Z 1298.265,A -85,B 0,C 180,E1 16103.952,E2 16103.952} C_VEL
LIN {X 0,Y 430.716,Z 1301.328,A -85,B 0,C 180,E1 16107.993,E2 16107.993} C_VEL
LIN {X 0,Y 430.785,Z 1300.837,A -85,B 0,C 180,E1 16112.025,E2 16112.025} C_VEL
LIN {X 0,Y 430.879,Z 1294.999,A -85,B 0,C 180,E1 16117.08,E2 16117.08} C_VEL
LIN {X 0,Y 430.876,Z 1294.88,A -85,B 0,C 180,E1 16117.142,E2 16117.142} C_VEL
LIN {X 0,Y 426.996,Z 1290.303,A -85,B 0,C 180,E1 16119.341,E2 16119.341} C_VEL
LIN {X 0,Y 423.389,Z 1284.648,A -85,B 0,C 180,E1 16121.541,E2 16121.541} C_VEL
LIN {X 0,Y 424.828,Z 1268.65,A -85,B 0,C 180,E1 16126.296,E2 16126.296} C_VEL
LIN {X 0,Y 427.538,Z 1247.579,A -85,B 0,C 180,E1 16130.768,E2 16130.768} C_VEL
LIN {X 0,Y 431.676,Z 1221.165,A -85,B 0,C 180,E1 16134.922,E2 16134.922} C_VEL
LIN {X 0,Y 439.529,Z 1176.943,A -85,B 0,C 180,E1 16140.059,E2 16140.059} C_VEL
LIN {X 0,Y 446.837,Z 1140.174,A -85,B 0,C 180,E1 16143.288,E2 16143.288} C_VEL
LIN {X 0,Y 454.214,Z 1100.508,A -85,B 0,C 180,E1 16145.803,E2 16145.803} C_VEL
LIN {X 0,Y 458.304,Z 1072.66,A -85,B 0,C 180,E1 16147.151,E2 16147.151} C_VEL
LIN {X 0,Y 454.228,Z 1045.141,A -85,B 0,C 180,E1 16149.159,E2 16149.159} C_VEL
LIN {X 0,Y 445.62,Z 1021.775,A -85,B 0,C 180,E1 16151.67,E2 16151.67} C_VEL
LIN {X 0,Y 436.235,Z 1002.884,A -85,B 0,C 180,E1 16154.622,E2 16154.622} C_VEL
LIN {X 0,Y 428.829,Z 990.899,A -85,B 0,C 180,E1 16157.631,E2 16157.631} C_VEL
LIN {X 0,Y 425.141,Z 984.689,A -85,B 0,C 180,E1 16159.774,E2 16159.774} C_VEL
LIN {X 0,Y 420.578,Z 978.144,A -85,B 0,C 180,E1 16164.977,E2 16164.977} C_VEL
LIN {X 0,Y 420.803,Z 978.677,A -85,B 0,C 180,E1 16167.956,E2 16167.956} C_VEL
LIN {X 0,Y 426.112,Z 985.826,A -85,B 0,C 180,E1 16173.196,E2 16173.196} C_VEL
LIN {X 0,Y 430.066,Z 991.607,A -85,B 0,C 180,E1 16175.384,E2 16175.384} C_VEL
LIN {X 0,Y 438.28,Z 1006.522,A -85,B 0,C 180,E1 16179.008,E2 16179.008} C_VEL
LIN {X 0,Y 446.986,Z 1024.67,A -85,B 0,C 180,E1 16182.084,E2 16182.084} C_VEL
LIN {X 0,Y 454.638,Z 1046.734,A -85,B 0,C 180,E1 16184.662,E2 16184.662} C_VEL
LIN {X 0,Y 453.149,Z 1060.644,A -85,B 0,C 180,E1 16185.325,E2 16185.325} C_VEL
LIN {X 0,Y 448.17,Z 1098.812,A -85,B 0,C 180,E1 16187.196,E2 16187.196} C_VEL
LIN {X 0,Y 443.406,Z 1127.135,A -85,B 0,C 180,E1 16189.431,E2 16189.431} C_VEL
LIN {X 0,Y 438.073,Z 1151.396,A -85,B 0,C 180,E1 16192.312,E2 16192.312} C_VEL
LIN {X 0,Y 433.449,Z 1170.039,A -85,B 0,C 180,E1 16195.591,E2 16195.591} C_VEL
LIN {X 0,Y 429.413,Z 1184.49,A -85,B 0,C 180,E1 16199.509,E2 16199.509} C_VEL
LIN {X 0,Y 426.878,Z 1192.101,A -85,B 0,C 180,E1 16203.066,E2 16203.066} C_VEL
LIN {X 0,Y 425.457,Z 1195.06,A -85,B 0,C 180,E1 16206.147,E2 16206.147} C_VEL
LIN {X 0,Y 424.662,Z 1194.094,A -85,B 0,C 180,E1 16210.291,E2 16210.291} C_VEL
LIN {X 0,Y 424.894,Z 1187.194,A -85,B 0,C 180,E1 16214.469,E2 16214.469} C_VEL
LIN {X 0,Y 425.822,Z 1174.664,A -85,B 0,C 180,E1 16218.423,E2 16218.423} C_VEL
LIN {X 0,Y 427.418,Z 1157.616,A -85,B 0,C 180,E1 16221.867,E2 16221.867} C_VEL
LIN {X 0,Y 429.772,Z 1134.591,A -85,B 0,C 180,E1 16225.042,E2 16225.042} C_VEL
LIN {X 0,Y 432.17,Z 1107.824,A -85,B 0,C 180,E1 16227.545,E2 16227.545} C_VEL
LIN {X 0,Y 434.232,Z 1077.852,A -85,B 0,C 180,E1 16229.354,E2 16229.354} C_VEL
LIN {X 0,Y 435.688,Z 1030.533,A -85,B 0,C 180,E1 16230.91,E2 16230.91} C_VEL
LIN {X 0,Y 420.822,Z 977.53,A -85,B 0,C 180,E1 16233.279,E2 16233.279} C_VEL
LIN {X 0,Y 420.531,Z 977.53,A -85,B 0,C 180,E1 16240.448,E2 16240.448} C_VEL
LIN {X 0,Y 420.445,Z 977.53,A -85,B 0,C 180,E1 16246.771,E2 16246.771} C_VEL
LIN {X 0,Y 420.534,Z 977.53,A -85,B 0,C 180,E1 16252.454,E2 16252.454} C_VEL
LIN {X 0,Y 420.754,Z 977.53,A -85,B 0,C 180,E1 16259.712,E2 16259.712} C_VEL
LIN {X 0,Y 421.087,Z 977.53,A -85,B 0,C 180,E1 16266.672,E2 16266.672} C_VEL
LIN {X 0,Y 421.391,Z 977.53,A -85,B 0,C 180,E1 16273.272,E2 16273.272} C_VEL
LIN {X 0,Y 421.717,Z 977.53,A -85,B 0,C 180,E1 16279.641,E2 16279.641} C_VEL
LIN {X 0,Y 422.182,Z 977.53,A -85,B 0,C 180,E1 16285.874,E2 16285.874} C_VEL
LIN {X 0,Y 422.35,Z 977.53,A -85,B 0,C 180,E1 16292.046,E2 16292.046} C_VEL
LIN {X 0,Y 421.832,Z 977.53,A -85,B 0,C 180,E1 16298.251,E2 16298.251} C_VEL
LIN {X 0,Y 421.484,Z 977.53,A -85,B 0,C 180,E1 16304.566,E2 16304.566} C_VEL
LIN {X 0,Y 421.177,Z 977.53,A -85,B 0,C 180,E1 16311.076,E2 16311.076} C_VEL
LIN {X 0,Y 420.844,Z 977.53,A -85,B 0,C 180,E1 16317.898,E2 16317.898} C_VEL
LIN {X 0,Y 420.592,Z 977.53,A -85,B 0,C 180,E1 16325.188,E2 16325.188} C_VEL
LIN {X 0,Y 420.499,Z 977.53,A -85,B 0,C 180,E1 16330.808,E2 16330.808} C_VEL
LIN {X 0,Y 420.423,Z 977.53,A -85,B 0,C 180,E1 16336.767,E2 16336.767} C_VEL
LIN {X 0,Y 420.596,Z 978.136,A -85,B 0,C 180,E1 16340.169,E2 16340.169} C_VEL
LIN {X 0,Y 441.849,Z 1033.009,A -85,B 0,C 180,E1 16343.269,E2 16343.269} C_VEL
LIN {X 0,Y 451.127,Z 1063.233,A -85,B 0,C 180,E1 16345.228,E2 16345.228} C_VEL
LIN {X 0,Y 446.197,Z 1102.636,A -85,B 0,C 180,E1 16347.426,E2 16347.426} C_VEL
LIN {X 0,Y 440.302,Z 1140.981,A -85,B 0,C 180,E1 16350.479,E2 16350.479} C_VEL
LIN {X 0,Y 434.851,Z 1173.395,A -85,B 0,C 180,E1 16354.027,E2 16354.027} C_VEL
LIN {X 0,Y 430.253,Z 1200.622,A -85,B 0,C 180,E1 16358.013,E2 16358.013} C_VEL
LIN {X 0,Y 426.712,Z 1223.08,A -85,B 0,C 180,E1 16362.419,E2 16362.419} C_VEL
LIN {X 0,Y 424.368,Z 1240.378,A -85,B 0,C 180,E1 16367.092,E2 16367.092} C_VEL
LIN {X 0,Y 423.264,Z 1252.182,A -85,B 0,C 180,E1 16371.753,E2 16371.753} C_VEL
LIN {X 0,Y 422.789,Z 1258.714,A -85,B 0,C 180,E1 16375.875,E2 16375.875} C_VEL
LIN {X 0,Y 422.803,Z 1261.618,A -85,B 0,C 180,E1 16379.985,E2 16379.985} C_VEL
LIN {X 0,Y 423.004,Z 1261.217,A -85,B 0,C 180,E1 16384.093,E2 16384.093} C_VEL
LIN {X 0,Y 423.987,Z 1255.959,A -85,B 0,C 180,E1 16389.239,E2 16389.239} C_VEL
LIN {X 0,Y 426.04,Z 1245.288,A -85,B 0,C 180,E1 16394.399,E2 16394.399} C_VEL
LIN {X 0,Y 430.175,Z 1228.553,A -85,B 0,C 180,E1 16399.532,E2 16399.532} C_VEL
LIN {X 0,Y 436.127,Z 1206.002,A -85,B 0,C 180,E1 16404.348,E2 16404.348} C_VEL
LIN {X 0,Y 443.563,Z 1178.993,A -85,B 0,C 180,E1 16408.552,E2 16408.552} C_VEL
LIN {X 0,Y 452.505,Z 1145.685,A -85,B 0,C 180,E1 16412.376,E2 16412.376} C_VEL
LIN {X 0,Y 462.07,Z 1107.339,A -85,B 0,C 180,E1 16415.575,E2 16415.575} C_VEL
LIN {X 0,Y 470.791,Z 1066.699,A -85,B 0,C 180,E1 16418.078,E2 16418.078} C_VEL
LIN {X 0,Y 469.139,Z 1051.624,A -85,B 0,C 180,E1 16420.05,E2 16420.05} C_VEL
LIN {X 0,Y 467.345,Z 1043.872,A -85,B 0,C 180,E1 16421.792,E2 16421.792} C_VEL
LIN {X 0,Y 466.475,Z 1038.203,A -85,B 0,C 180,E1 16424.399,E2 16424.399} C_VEL
LIN {X 0,Y 466.527,Z 1040.14,A -85,B 0,C 180,E1 16425.898,E2 16425.898} C_VEL
LIN {X 0,Y 468.452,Z 1045.979,A -85,B 0,C 180,E1 16428.043,E2 16428.043} C_VEL
LIN {X 0,Y 469.426,Z 1051.419,A -85,B 0,C 180,E1 16428.995,E2 16428.995} C_VEL
LIN {X 0,Y 469.105,Z 1080.536,A -85,B 0,C 180,E1 16431.519,E2 16431.519} C_VEL
LIN {X 0,Y 459.401,Z 1123.908,A -85,B 0,C 180,E1 16433.761,E2 16433.761} C_VEL
LIN {X 0,Y 449.945,Z 1163.625,A -85,B 0,C 180,E1 16436.688,E2 16436.688} C_VEL
LIN {X 0,Y 441.253,Z 1199.598,A -85,B 0,C 180,E1 16440.289,E2 16440.289} C_VEL
LIN {X 0,Y 433.98,Z 1230.311,A -85,B 0,C 180,E1 16444.411,E2 16444.411} C_VEL
LIN {X 0,Y 428.473,Z 1255.843,A -85,B 0,C 180,E1 16449.029,E2 16449.029} C_VEL
LIN {X 0,Y 424.98,Z 1275.746,A -85,B 0,C 180,E1 16453.971,E2 16453.971} C_VEL
LIN {X 0,Y 423.276,Z 1290.12,A -85,B 0,C 180,E1 16459.177,E2 16459.177} C_VEL
LIN {X 0,Y 422.88,Z 1297.953,A -85,B 0,C 180,E1 16463.839,E2 16463.839} C_VEL
LIN {X 0,Y 422.839,Z 1300.939,A -85,B 0,C 180,E1 16467.956,E2 16467.956} C_VEL
LIN {X 0,Y 422.897,Z 1300.368,A -85,B 0,C 180,E1 16472.063,E2 16472.063} C_VEL
LIN {X 0,Y 422.982,Z 1294.387,A -85,B 0,C 180,E1 16477.212,E2 16477.212} C_VEL
LIN {X 0,Y 423.389,Z 1284.648,A -85,B 0,C 180,E1 16481.541,E2 16481.541} C_VEL
LIN {X 0,Y 422.41,Z 1281.497,A -85,B 0,C 180,E1 16482.639,E2 16482.639} C_VEL
LIN {X 0,Y 416.758,Z 1271.634,A -85,B 0,C 180,E1 16485.571,E2 16485.571} C_VEL
LIN {X 0,Y 416.754,Z 1270.596,A -85,B 0,C 180,E1 16485.839,E2 16485.839} C_VEL
LIN {X 0,Y 419.441,Z 1249.699,A -85,B 0,C 180,E1 16490.511,E2 16490.511} C_VEL
LIN {X 0,Y 423.626,Z 1223.267,A -85,B 0,C 180,E1 16494.852,E2 16494.852} C_VEL
LIN {X 0,Y 432.188,Z 1179.054,A -85,B 0,C 180,E1 16500.364,E2 16500.364} C_VEL
LIN {X 0,Y 440.258,Z 1140.776,A -85,B 0,C 180,E1 16503.848,E2 16503.848} C_VEL
LIN {X 0,Y 448.313,Z 1099.803,A -85,B 0,C 180,E1 16506.499,E2 16506.499} C_VEL
LIN {X 0,Y 452.263,Z 1074.345,A -85,B 0,C 180,E1 16507.773,E2 16507.773} C_VEL
LIN {X 0,Y 448.814,Z 1048.572,A -85,B 0,C 180,E1 16509.757,E2 16509.757} C_VEL
LIN {X 0,Y 440.573,Z 1025.146,A -85,B 0,C 180,E1 16512.435,E2 16512.435} C_VEL
LIN {X 0,Y 431.745,Z 1007.447,A -85,B 0,C 180,E1 16515.497,E2 16515.497} C_VEL
LIN {X 0,Y 425.972,Z 997.819,A -85,B 0,C 180,E1 16518.057,E2 16518.057} C_VEL
LIN {X 0,Y 422.57,Z 992.021,A -85,B 0,C 180,E1 16520.147,E2 16520.147} C_VEL
LIN {X 0,Y 418.595,Z 985.284,A -85,B 0,C 180,E1 16525.795,E2 16525.795} C_VEL
LIN {X 0,Y 419.105,Z 987.845,A -85,B 0,C 180,E1 16528.987,E2 16528.987} C_VEL
LIN {X 0,Y 423.426,Z 993.375,A -85,B 0,C 180,E1 16532.997,E2 16532.997} C_VEL
LIN {X 0,Y 427.717,Z 1000.665,A -85,B 0,C 180,E1 16535.588,E2 16535.588} C_VEL
LIN {X 0,Y 434.868,Z 1013.68,A -85,B 0,C 180,E1 16538.835,E2 16538.835} C_VEL
LIN {X 0,Y 443.003,Z 1031.865,A -85,B 0,C 180,E1 16541.917,E2 16541.917} C_VEL
LIN {X 0,Y 449.035,Z 1050.655,A -85,B 0,C 180,E1 16544.16,E2 16544.16} C_VEL
LIN {X 0,Y 442.131,Z 1098.809,A -85,B 0,C 180,E1 16546.514,E2 16546.514} C_VEL
LIN {X 0,Y 437.309,Z 1125.988,A -85,B 0,C 180,E1 16548.65,E2 16548.65} C_VEL
LIN {X 0,Y 431.855,Z 1150.039,A -85,B 0,C 180,E1 16551.44,E2 16551.44} C_VEL
LIN {X 0,Y 426.574,Z 1170.221,A -85,B 0,C 180,E1 16554.937,E2 16554.937} C_VEL
LIN {X 0,Y 422.131,Z 1185.131,A -85,B 0,C 180,E1 16558.986,E2 16558.986} C_VEL
LIN {X 0,Y 419.058,Z 1193.636,A -85,B 0,C 180,E1 16563.124,E2 16563.124} C_VEL
LIN {X 0,Y 417.586,Z 1196.258,A -85,B 0,C 180,E1 16566.264,E2 16566.264} C_VEL
LIN {X 0,Y 416.824,Z 1194.784,A -85,B 0,C 180,E1 16570.486,E2 16570.486} C_VEL
LIN {X 0,Y 417.077,Z 1187.39,A -85,B 0,C 180,E1 16574.747,E2 16574.747} C_VEL
LIN {X 0,Y 418.092,Z 1174.279,A -85,B 0,C 180,E1 16578.776,E2 16578.776} C_VEL
LIN {X 0,Y 420.015,Z 1155.17,A -85,B 0,C 180,E1 16582.533,E2 16582.533} C_VEL
LIN {X 0,Y 422.36,Z 1131.737,A -85,B 0,C 180,E1 16585.633,E2 16585.633} C_VEL
LIN {X 0,Y 424.798,Z 1105.132,A -85,B 0,C 180,E1 16588.038,E2 16588.038} C_VEL
LIN {X 0,Y 426.888,Z 1074.269,A -85,B 0,C 180,E1 16589.81,E2 16589.81} C_VEL
LIN {X 0,Y 427.865,Z 1030.811,A -85,B 0,C 180,E1 16591.243,E2 16591.243} C_VEL
LIN {X 0,Y 412.87,Z 977.53,A -85,B 0,C 180,E1 16593.701,E2 16593.701} C_VEL
LIN {X 0,Y 412.566,Z 977.53,A -85,B 0,C 180,E1 16601.398,E2 16601.398} C_VEL
LIN {X 0,Y 412.51,Z 977.53,A -85,B 0,C 180,E1 16608.596,E2 16608.596} C_VEL
LIN {X 0,Y 412.581,Z 977.53,A -85,B 0,C 180,E1 16614,E2 16614} C_VEL
LIN {X 0,Y 412.75,Z 977.53,A -85,B 0,C 180,E1 16619.061,E2 16619.061} C_VEL
LIN {X 0,Y 413.12,Z 977.53,A -85,B 0,C 180,E1 16626.194,E2 16626.194} C_VEL
LIN {X 0,Y 413.431,Z 977.53,A -85,B 0,C 180,E1 16632.94,E2 16632.94} C_VEL
LIN {X 0,Y 413.778,Z 977.53,A -85,B 0,C 180,E1 16639.44,E2 16639.44} C_VEL
LIN {X 0,Y 414.265,Z 977.53,A -85,B 0,C 180,E1 16645.795,E2 16645.795} C_VEL
LIN {X 0,Y 414.439,Z 977.53,A -85,B 0,C 180,E1 16652.086,E2 16652.086} C_VEL
LIN {X 0,Y 413.869,Z 977.53,A -85,B 0,C 180,E1 16658.632,E2 16658.632} C_VEL
